legal notes
=================
| SPDX-FileCopyrightText: © 2022 ekvip automation GmbH <info@ekvip.de>
| SPDX-License-Identifier: Apache-2.0
| For details check: Apache-2.0_

.. _Apache-2.0: https://www.apache.org/licenses/LICENSE-2.0

.. </legal notes>



*)

METHOD orMaskIsEqualTo
VAR_INPUT
	(* current value to check *)
	currentValue	:__XWORD;
	(* 2nd operand for bitwise operation *)
	mask			:__XWORD;
	(* expected result after masking *)
	expectedValue	:__XWORD;
	(* message if the assertion is false *)
	message			:AssertMessage;
END_VAR
END_METHOD

(*

## Short summary
This assertion method checks if the result current value bitwise ``OR`` mask 
is not equal to the unexpected value

.. <legal notes>

legal notes
=================
| SPDX-FileCopyrightText: © 2022 ekvip automation GmbH <info@ekvip.de>
| SPDX-License-Identifier: Apache-2.0
| For details check: Apache-2.0_

.. _Apache-2.0: https://www.apache.org/licenses/LICENSE-2.0

.. </legal notes>



*)

METHOD orMaskIsNotEqualTo
VAR_INPUT
	(* current value to check *)
	currentValue	:__XWORD;
	(* 2nd operand for bitwise operation *)
	mask			:__XWORD;
	(* unexpected result after masking *)
	unexpectedValue	:__XWORD;
	(* message if the assertion is false *)
	message			:AssertMessage;
END_VAR
END_METHOD

(*

## Short summary
This assertion method checks if the current value is equal to the expected value

.. <legal notes>

legal notes
=================
| SPDX-FileCopyrightText: © 2022 ekvip automation GmbH <info@ekvip.de>
| SPDX-License-Identifier: Apache-2.0
| For details check: Apache-2.0_

.. _Apache-2.0: https://www.apache.org/licenses/LICENSE-2.0

.. </legal notes>



*)

METHOD valueIsEqualTo
VAR_INPUT
	(* current value to check *)
	currentValue	:__XWORD;
	(* expected value to compare *)
	expectedValue	:__XWORD;
	(* message if the assertion is false *)
	message			:AssertMessage;
END_VAR
END_METHOD

(*

## Short summary
This assertion method checks if the current value is greater than the less value

.. <legal notes>

legal notes
=================
| SPDX-FileCopyrightText: © 2022 ekvip automation GmbH <info@ekvip.de>
| SPDX-License-Identifier: Apache-2.0
| For details check: Apache-2.0_

.. _Apache-2.0: https://www.apache.org/licenses/LICENSE-2.0

.. </legal notes>



*)

METHOD valueIsGreaterThan
VAR_INPUT
	(* current value to check *)
	currentValue	:__XWORD;
	(* less than lower limit *)
	lessValue		:__XWORD;
	(* message if the assertion is false *)
	message			:AssertMessage;
END_VAR
END_METHOD

(*

## Short summary
This assertion method checks if the current value is inside a limit

**Attention:** 
	limits are included: ``valueIsInRangeOf(3, 3, 3)`` is a true assertion

.. <legal notes>

legal notes
=================
| SPDX-FileCopyrightText: © 2022 ekvip automation GmbH <info@ekvip.de>
| SPDX-License-Identifier: Apache-2.0
| For details check: Apache-2.0_

.. _Apache-2.0: https://www.apache.org/licenses/LICENSE-2.0

.. </legal notes>



*)

METHOD valueIsInRangeOf
VAR_INPUT
	(* lower limit for the current value *)
	lowerLimit		:__XWORD;
	(* current value to check *)
	currentValue	:__XWORD;
	(* upper limit for the current value *)
	upperLimit		:__XWORD;
	(* message if the assertion is false *)
	message			:AssertMessage;
END_VAR
END_METHOD

(*

## Short summary
This assertion method checks if the current value is less than the greater value

.. <legal notes>

legal notes
=================
| SPDX-FileCopyrightText: © 2022 ekvip automation GmbH <info@ekvip.de>
| SPDX-License-Identifier: Apache-2.0
| For details check: Apache-2.0_

.. _Apache-2.0: https://www.apache.org/licenses/LICENSE-2.0

.. </legal notes>



*)

METHOD valueIsLessThan
VAR_INPUT
	(* current value to check *)
	currentValue	:__XWORD;
	(* greater than upper limit *)
	greaterValue	:__XWORD;
	(* message if the assertion is false *)
	message			:AssertMessage;
END_VAR
END_METHOD

(*

## Short summary
This assertion method checks if the current value is less than or equal to the maximum value

.. <legal notes>

legal notes
=================
| SPDX-FileCopyrightText: © 2022 ekvip automation GmbH <info@ekvip.de>
| SPDX-License-Identifier: Apache-2.0
| For details check: Apache-2.0_

.. _Apache-2.0: https://www.apache.org/licenses/LICENSE-2.0

.. </legal notes>



*)

METHOD valueIsMax
VAR_INPUT
	(* current value to check *)
	currentValue	:__XWORD;
	(* upper limit for the current value *)
	maximumValue	:__XWORD;
	(* message if the assertion is false *)
	message			:AssertMessage;
END_VAR
END_METHOD

(*

## Short summary
This assertion method checks if the current value is greater than or equal to the minimum value

.. <legal notes>

legal notes
=================
| SPDX-FileCopyrightText: © 2022 ekvip automation GmbH <info@ekvip.de>
| SPDX-License-Identifier: Apache-2.0
| For details check: Apache-2.0_

.. _Apache-2.0: https://www.apache.org/licenses/LICENSE-2.0

.. </legal notes>



*)

METHOD valueIsMin
VAR_INPUT
	(* current value to check *)
	currentValue	:__XWORD;
	(* lower limit for the current value *)
	minimumValue	:__XWORD;
	(* message if the assertion is false *)
	message			:AssertMessage;
END_VAR
END_METHOD

(*

## Short summary
This assertion method checks if the current value is not equal to the unexpected value

.. <legal notes>

legal notes
=================
| SPDX-FileCopyrightText: © 2022 ekvip automation GmbH <info@ekvip.de>
| SPDX-License-Identifier: Apache-2.0
| For details check: Apache-2.0_

.. _Apache-2.0: https://www.apache.org/licenses/LICENSE-2.0

.. </legal notes>



*)

METHOD valueIsNotEqualTo
VAR_INPUT
	(* current value to check *)
	currentValue	:__XWORD;
	(* unexpected value to compare *)
	unexpectedValue	:__XWORD;
	(* message if the assertion is false *)
	message			:AssertMessage;
END_VAR
END_METHOD

(*

## Short summary
This assertion method checks if the result current value bitwise ``XOR`` mask is equal to the expected value

.. <legal notes>

legal notes
=================
| SPDX-FileCopyrightText: © 2022 ekvip automation GmbH <info@ekvip.de>
| SPDX-License-Identifier: Apache-2.0
| For details check: Apache-2.0_

.. _Apache-2.0: https://www.apache.org/licenses/LICENSE-2.0

.. </legal notes>



*)

METHOD xorMaskIsEqualTo
VAR_INPUT
	(* current value to check *)
	currentValue	:__XWORD;
	(* 2nd operand for bitwise operation *)
	mask			:__XWORD;
	(* expected result after masking *)
	expectedValue	:__XWORD;
	(* message if the assertion is false *)
	message			:AssertMessage;
END_VAR
END_METHOD

(*

## Short summary
This assertion method checks if the result current value bitwise ``XOR`` mask 
is not equal to the unexpected value

.. <legal notes>

legal notes
=================
| SPDX-FileCopyrightText: © 2022 ekvip automation GmbH <info@ekvip.de>
| SPDX-License-Identifier: Apache-2.0
| For details check: Apache-2.0_

.. _Apache-2.0: https://www.apache.org/licenses/LICENSE-2.0

.. </legal notes>



*)

METHOD xorMaskIsNotEqualTo
VAR_INPUT
	(* current value to check *)
	currentValue	:__XWORD;
	(* 2nd operand for bitwise operation *)
	mask			:__XWORD;
	(* unexpected result after masking *)
	unexpectedValue	:__XWORD;
	(* message if the assertion is false *)
	message			:AssertMessage;
END_VAR
END_METHOD

END_INTERFACE

// ---- Assertor/Assertions/BooleanAssertion/interfaces/IBooleanAssertion.TcIO
(*

## Short summary
This interface provides assert statements for booleans 

.. <legal notes>

legal notes
=================
| SPDX-FileCopyrightText: © 2022 ekvip automation GmbH <info@ekvip.de>
| SPDX-License-Identifier: Apache-2.0
| For details check: Apache-2.0_

.. _Apache-2.0: https://www.apache.org/licenses/LICENSE-2.0

.. </legal notes>



*)

INTERFACE IBooleanAssertion EXTENDS __SYSTEM.IQueryInterface

(*

## Short summary
This assertion method checks if the current value is equal to the expected value

.. <legal notes>

legal notes
=================
| SPDX-FileCopyrightText: © 2022 ekvip automation GmbH <info@ekvip.de>
| SPDX-License-Identifier: Apache-2.0
| For details check: Apache-2.0_

.. _Apache-2.0: https://www.apache.org/licenses/LICENSE-2.0

.. </legal notes>



*)

METHOD valueIsEqualTo
VAR_INPUT
	(* current value to check *)
	currentValue	:BOOL;
	(* expected value to compare *)
	expectedValue	:BOOL;
	(* message if the assertion is false *)
	message			:AssertMessage;
END_VAR
END_METHOD

(*

## Short summary
This assertion method checks if the current value is ``FALSE``

.. <legal notes>

legal notes
=================
| SPDX-FileCopyrightText: © 2022 ekvip automation GmbH <info@ekvip.de>
| SPDX-License-Identifier: Apache-2.0
| For details check: Apache-2.0_

.. _Apache-2.0: https://www.apache.org/licenses/LICENSE-2.0

.. </legal notes>



*)

METHOD valueIsFalse
VAR_INPUT
	(* current value to check *)
	currentValue	:BOOL;
	(* message if the assertion is false *)
	message			:AssertMessage;
END_VAR
END_METHOD

(*

## Short summary
This assertion method checks if the current value is not equal to the unexpected value

.. <legal notes>

legal notes
=================
| SPDX-FileCopyrightText: © 2022 ekvip automation GmbH <info@ekvip.de>
| SPDX-License-Identifier: Apache-2.0
| For details check: Apache-2.0_

.. _Apache-2.0: https://www.apache.org/licenses/LICENSE-2.0

.. </legal notes>



*)

METHOD valueIsNotEqualTo
VAR_INPUT
	(* current value to check *)
	currentValue	:BOOL;
	(* unexpected value to compare *)
	unexpectedValue	:BOOL;
	(* message if the assertion is false *)
	message			:AssertMessage;
END_VAR
END_METHOD

(*

## Short summary
This assertion method checks if the current value is ``TRUE``

.. <legal notes>

legal notes
=================
| SPDX-FileCopyrightText: © 2022 ekvip automation GmbH <info@ekvip.de>
| SPDX-License-Identifier: Apache-2.0
| For details check: Apache-2.0_

.. _Apache-2.0: https://www.apache.org/licenses/LICENSE-2.0

.. </legal notes>



*)

METHOD valueIsTrue
VAR_INPUT
	(* current value to check *)
	currentValue	:BOOL;
	(* message if the assertion is false *)
	message			:AssertMessage;
END_VAR
END_METHOD

END_INTERFACE

// ---- Assertor/Assertions/DateAndTimeAssertions/32Bit/Date/interfaces/I32BitDateAssertions.TcIO
(*

## Short summary
This interface provides assert statements for 32 bit ``DATE``  

.. <legal notes>

legal notes
=================
| SPDX-FileCopyrightText: © 2022 ekvip automation GmbH <info@ekvip.de>
| SPDX-License-Identifier: Apache-2.0
| For details check: Apache-2.0_

.. _Apache-2.0: https://www.apache.org/licenses/LICENSE-2.0

.. </legal notes>



*)

INTERFACE I32BitDateAssertions EXTENDS __SYSTEM.IQueryInterface

(*

## Short summary
This assertion method checks if the current value is equal to the expected value

.. <legal notes>

legal notes
=================
| SPDX-FileCopyrightText: © 2022 ekvip automation GmbH <info@ekvip.de>
| SPDX-License-Identifier: Apache-2.0
| For details check: Apache-2.0_

.. _Apache-2.0: https://www.apache.org/licenses/LICENSE-2.0

.. </legal notes>



*)

METHOD valueIsEqualTo
VAR_INPUT
	(* current value to check *)
	currentValue	:DATE;
	(* expected value to compare *)
	expectedValue	:DATE;
	(* message if the assertion is false *)
	message			:AssertMessage;
END_VAR
END_METHOD

(*

## Short summary
This assertion method checks if the current value is greater than the less value

.. <legal notes>

legal notes
=================
| SPDX-FileCopyrightText: © 2022 ekvip automation GmbH <info@ekvip.de>
| SPDX-License-Identifier: Apache-2.0
| For details check: Apache-2.0_

.. _Apache-2.0: https://www.apache.org/licenses/LICENSE-2.0

.. </legal notes>



*)

METHOD valueIsGreaterThan
VAR_INPUT
	(* current value to check *)
	currentValue	:DATE;
	(* less than lower limit *)
	lessValue		:DATE;
	(* message if the assertion is false *)
	message			:AssertMessage;
END_VAR
END_METHOD

(*

## Short summary
This assertion method checks if the current value is inside a limit

**Attention:** 
	limits are included: ``valueIsInRangeOf(date#1970-01-01, date#1970-01-01, date#1970-01-01)``
	is a true assertion

.. <legal notes>

legal notes
=================
| SPDX-FileCopyrightText: © 2022 ekvip automation GmbH <info@ekvip.de>
| SPDX-License-Identifier: Apache-2.0
| For details check: Apache-2.0_

.. _Apache-2.0: https://www.apache.org/licenses/LICENSE-2.0

.. </legal notes>



*)

METHOD valueIsInRangeOf
VAR_INPUT
	(* lower limit for the current value *)
	lowerLimit		:DATE;
	(* current value to check *)
	currentValue	:DATE;
	(* upper limit for the current value *)
	upperLimit		:DATE;
	(* message if the assertion is false *)
	message			:AssertMessage;
END_VAR
END_METHOD

(*

## Short summary
This assertion method checks if the current value is less than the greater value

.. <legal notes>

legal notes
=================
| SPDX-FileCopyrightText: © 2022 ekvip automation GmbH <info@ekvip.de>
| SPDX-License-Identifier: Apache-2.0
| For details check: Apache-2.0_

.. _Apache-2.0: https://www.apache.org/licenses/LICENSE-2.0

.. </legal notes>



*)

METHOD valueIsLessThan
VAR_INPUT
	(* current value to check *)
	currentValue	:DATE;
	(* greater than upper limit *)
	greaterValue	:DATE;
	(* message if the assertion is false *)
	message			:AssertMessage;
END_VAR
END_METHOD

(*

## Short summary
This assertion method checks if the current value is less than or equal to the maximum value

.. <legal notes>

legal notes
=================
| SPDX-FileCopyrightText: © 2022 ekvip automation GmbH <info@ekvip.de>
| SPDX-License-Identifier: Apache-2.0
| For details check: Apache-2.0_

.. _Apache-2.0: https://www.apache.org/licenses/LICENSE-2.0

.. </legal notes>



*)

METHOD valueIsMax
VAR_INPUT
	(* current value to check *)
	currentValue	:DATE;
	(* upper limit for the current value *)
	maximumValue	:DATE;
	(* message if the assertion is false *)
	message			:AssertMessage;
END_VAR
END_METHOD

(*

## Short summary
This assertion method checks if the current value is greater than or equal to the minimum value

.. <legal notes>

legal notes
=================
| SPDX-FileCopyrightText: © 2022 ekvip automation GmbH <info@ekvip.de>
| SPDX-License-Identifier: Apache-2.0
| For details check: Apache-2.0_

.. _Apache-2.0: https://www.apache.org/licenses/LICENSE-2.0

.. </legal notes>



*)

METHOD valueIsMin
VAR_INPUT
	(* current value to check *)
	currentValue	:DATE;
	(* lower limit for the current value *)
	minimumValue	:DATE;
	(* message if the assertion is false *)
	message			:AssertMessage;
END_VAR
END_METHOD

(*

## Short summary
This assertion method checks if the current value is not equal to the unexpected value

.. <legal notes>

legal notes
=================
| SPDX-FileCopyrightText: © 2022 ekvip automation GmbH <info@ekvip.de>
| SPDX-License-Identifier: Apache-2.0
| For details check: Apache-2.0_

.. _Apache-2.0: https://www.apache.org/licenses/LICENSE-2.0

.. </legal notes>



*)

METHOD valueIsNotEqualTo
VAR_INPUT
	(* current value to check *)
	currentValue	:DATE;
	(* unexpected value to compare *)
	unexpectedValue	:DATE;
	(* message if the assertion is false *)
	message			:AssertMessage;
END_VAR
END_METHOD

END_INTERFACE

// ---- Assertor/Assertions/DateAndTimeAssertions/32Bit/DT/interfaces/I32BitDtAssertions.TcIO
(*

## Short summary
This interface provides assert statements for 32 bit date and time ``DT``  

.. <legal notes>

legal notes
=================
| SPDX-FileCopyrightText: © 2022 ekvip automation GmbH <info@ekvip.de>
| SPDX-License-Identifier: Apache-2.0
| For details check: Apache-2.0_

.. _Apache-2.0: https://www.apache.org/licenses/LICENSE-2.0

.. </legal notes>



*)

INTERFACE I32BitDtAssertions EXTENDS __SYSTEM.IQueryInterface

(*

## Short summary
This assertion method checks if the current value is equal to the expected value

.. <legal notes>

legal notes
=================
| SPDX-FileCopyrightText: © 2022 ekvip automation GmbH <info@ekvip.de>
| SPDX-License-Identifier: Apache-2.0
| For details check: Apache-2.0_

.. _Apache-2.0: https://www.apache.org/licenses/LICENSE-2.0

.. </legal notes>



*)

METHOD valueIsEqualTo
VAR_INPUT
	(* current value to check *)
	currentValue	:DT;
	(* expected value to compare *)
	expectedValue	:DT;
	(* message if the assertion is false *)
	message			:AssertMessage;
END_VAR
END_METHOD

(*

## Short summary
This assertion method checks if the current value is greater than the less value

.. <legal notes>

legal notes
=================
| SPDX-FileCopyrightText: © 2022 ekvip automation GmbH <info@ekvip.de>
| SPDX-License-Identifier: Apache-2.0
| For details check: Apache-2.0_

.. _Apache-2.0: https://www.apache.org/licenses/LICENSE-2.0

.. </legal notes>



*)

METHOD valueIsGreaterThan
VAR_INPUT
	(* current value to check *)
	currentValue	:DT;
	(* less than lower limit *)
	lessValue		:DT;
	(* message if the assertion is false *)
	message			:AssertMessage;
END_VAR
END_METHOD

(*

## Short summary
This assertion method checks if the current value is inside a limit

**Attention:** 
	limits are included: ``valueIsInRangeOf(dt#1970-01-01-0:0:0, dt#1970-01-01-0:0:0, dt#1970-01-01-0:0:0)``
	is a true assertion

.. <legal notes>

legal notes
=================
| SPDX-FileCopyrightText: © 2022 ekvip automation GmbH <info@ekvip.de>
| SPDX-License-Identifier: Apache-2.0
| For details check: Apache-2.0_

.. _Apache-2.0: https://www.apache.org/licenses/LICENSE-2.0

.. </legal notes>



*)

METHOD valueIsInRangeOf
VAR_INPUT
	(* lower limit for the current value *)
	lowerLimit		:DT;
	(* current value to check *)
	currentValue	:DT;
	(* upper limit for the current value *)
	upperLimit		:DT;
	(* message if the assertion is false *)
	message			:AssertMessage;
END_VAR
END_METHOD

(*

## Short summary
This assertion method checks if the current value is less than the greater value

.. <legal notes>

legal notes
=================
| SPDX-FileCopyrightText: © 2022 ekvip automation GmbH <info@ekvip.de>
| SPDX-License-Identifier: Apache-2.0
| For details check: Apache-2.0_

.. _Apache-2.0: https://www.apache.org/licenses/LICENSE-2.0

.. </legal notes>



*)

METHOD valueIsLessThan
VAR_INPUT
	(* current value to check *)
	currentValue	:DT;
	(* greater than upper limit *)
	greaterValue	:DT;
	(* message if the assertion is false *)
	message			:AssertMessage;
END_VAR
END_METHOD

(*

## Short summary
This assertion method checks if the current value is less than or equal to the maximum value

.. <legal notes>

legal notes
=================
| SPDX-FileCopyrightText: © 2022 ekvip automation GmbH <info@ekvip.de>
| SPDX-License-Identifier: Apache-2.0
| For details check: Apache-2.0_

.. _Apache-2.0: https://www.apache.org/licenses/LICENSE-2.0

.. </legal notes>



*)

METHOD valueIsMax
VAR_INPUT
	(* current value to check *)
	currentValue	:DT;
	(* upper limit for the current value *)
	maximumValue	:DT;
	(* message if the assertion is false *)
	message			:AssertMessage;
END_VAR
END_METHOD

(*

## Short summary
This assertion method checks if the current value is greater than or equal to the minimum value

.. <legal notes>

legal notes
=================
| SPDX-FileCopyrightText: © 2022 ekvip automation GmbH <info@ekvip.de>
| SPDX-License-Identifier: Apache-2.0
| For details check: Apache-2.0_

.. _Apache-2.0: https://www.apache.org/licenses/LICENSE-2.0

.. </legal notes>



*)

METHOD valueIsMin
VAR_INPUT
	(* current value to check *)
	currentValue	:DT;
	(* lower limit for the current value *)
	minimumValue	:DT;
	(* message if the assertion is false *)
	message			:AssertMessage;
END_VAR
END_METHOD

(*

## Short summary
This assertion method checks if the current value is not equal to the unexpected value

.. <legal notes>

legal notes
=================
| SPDX-FileCopyrightText: © 2022 ekvip automation GmbH <info@ekvip.de>
| SPDX-License-Identifier: Apache-2.0
| For details check: Apache-2.0_

.. _Apache-2.0: https://www.apache.org/licenses/LICENSE-2.0

.. </legal notes>



*)

METHOD valueIsNotEqualTo
VAR_INPUT
	(* current value to check *)
	currentValue	:DT;
	(* unexpected value to compare *)
	unexpectedValue	:DT;
	(* message if the assertion is false *)
	message			:AssertMessage;
END_VAR
END_METHOD

END_INTERFACE

// ---- Assertor/Assertions/DateAndTimeAssertions/32Bit/interfaces/ISimpleDateAndTimeAssertions.TcIO
(*

## Short summary

This interface provides assert statements for date and time types with 32 bit length
For date and time (``DT``) use `ISimpleDateAndTimeAssertions.dateAndTime`
For date (``DATE``) use  `ISimpleDateAndTimeAssertions.dateOnly`
For time of day (``TOD``) use  `ISimpleDateAndTimeAssertions.timeOfDay`

.. <legal notes>

legal notes
=================
| SPDX-FileCopyrightText: © 2022 ekvip automation GmbH <info@ekvip.de>
| SPDX-License-Identifier: Apache-2.0
| For details check: Apache-2.0_

.. _Apache-2.0: https://www.apache.org/licenses/LICENSE-2.0

.. </legal notes>



*)

INTERFACE ISimpleDateAndTimeAssertions EXTENDS __SYSTEM.IQueryInterface

(*

## Short summary
Returns the interface `I32BitDtAssertions` with assert statements for 32 bit date and time ``DT``

.. <legal notes>

legal notes
=================
| SPDX-FileCopyrightText: © 2022 ekvip automation GmbH <info@ekvip.de>
| SPDX-License-Identifier: Apache-2.0
| For details check: Apache-2.0_

.. _Apache-2.0: https://www.apache.org/licenses/LICENSE-2.0

.. </legal notes>

*)

PROPERTY dateAndTime :I32BitDtAssertions
GET
END_GET
END_PROPERTY

(*

## Short summary
Returns the interface `I32BitDateAssertions` with assert statements for 32 bit date ``DATE``

.. <legal notes>

legal notes
=================
| SPDX-FileCopyrightText: © 2022 ekvip automation GmbH <info@ekvip.de>
| SPDX-License-Identifier: Apache-2.0
| For details check: Apache-2.0_

.. _Apache-2.0: https://www.apache.org/licenses/LICENSE-2.0

.. </legal notes>

*)

PROPERTY dateOnly :I32BitDateAssertions
GET
END_GET
END_PROPERTY

(*

## Short summary
Returns the interface `I32BitTodAssertions` with assert statements for 32 bit time of day ``TOD``

.. <legal notes>

legal notes
=================
| SPDX-FileCopyrightText: © 2022 ekvip automation GmbH <info@ekvip.de>
| SPDX-License-Identifier: Apache-2.0
| For details check: Apache-2.0_

.. _Apache-2.0: https://www.apache.org/licenses/LICENSE-2.0

.. </legal notes>

*)

PROPERTY timeOfDay :I32BitTodAssertions
GET
END_GET
END_PROPERTY

END_INTERFACE

// ---- Assertor/Assertions/DateAndTimeAssertions/32Bit/TOD/interfaces/I32BitTodAssertions.TcIO
(*

## Short summary
This interface provides assert statements for 32 bit time of day ``TOD``  

.. <legal notes>

legal notes
=================
| SPDX-FileCopyrightText: © 2022 ekvip automation GmbH <info@ekvip.de>
| SPDX-License-Identifier: Apache-2.0
| For details check: Apache-2.0_

.. _Apache-2.0: https://www.apache.org/licenses/LICENSE-2.0

.. </legal notes>



*)

INTERFACE I32BitTodAssertions EXTENDS __SYSTEM.IQueryInterface

(*

## Short summary
This assertion method checks if the current value is equal to the expected value

.. <legal notes>

legal notes
=================
| SPDX-FileCopyrightText: © 2022 ekvip automation GmbH <info@ekvip.de>
| SPDX-License-Identifier: Apache-2.0
| For details check: Apache-2.0_

.. _Apache-2.0: https://www.apache.org/licenses/LICENSE-2.0

.. </legal notes>



*)

METHOD valueIsEqualTo
VAR_INPUT
	(* current value to check *)
	currentValue	:TOD;
	(* expected value to compare *)
	expectedValue	:TOD;
	(* message if the assertion is false *)
	message			:AssertMessage;
END_VAR
END_METHOD

(*

## Short summary
This assertion method checks if the current value is greater than the less value

.. <legal notes>

legal notes
=================
| SPDX-FileCopyrightText: © 2022 ekvip automation GmbH <info@ekvip.de>
| SPDX-License-Identifier: Apache-2.0
| For details check: Apache-2.0_

.. _Apache-2.0: https://www.apache.org/licenses/LICENSE-2.0

.. </legal notes>



*)

METHOD valueIsGreaterThan
VAR_INPUT
	(* current value to check *)
	currentValue	:TOD;
	(* less than lower limit *)
	lessValue		:TOD;
	(* message if the assertion is false *)
	message			:AssertMessage;
END_VAR
END_METHOD

(*

## Short summary
This assertion method checks if the current value is inside a limit

**Attention:** 
	limits are included: ``valueIsInRangeOf(tod#3:0:0, tod#3:0:0, tod#3:0:0)`` is a true assertion

.. <legal notes>

legal notes
=================
| SPDX-FileCopyrightText: © 2022 ekvip automation GmbH <info@ekvip.de>
| SPDX-License-Identifier: Apache-2.0
| For details check: Apache-2.0_

.. _Apache-2.0: https://www.apache.org/licenses/LICENSE-2.0

.. </legal notes>



*)

METHOD valueIsInRangeOf
VAR_INPUT
	(* lower limit for the current value *)
	lowerLimit		:TOD;
	(* current value to check *)
	currentValue	:TOD;
	(* upper limit for the current value *)
	upperLimit		:TOD;
	(* message if the assertion is false *)
	message			:AssertMessage;
END_VAR
END_METHOD

(*

## Short summary
This assertion method checks if the current value is less than the greater value

.. <legal notes>

legal notes
=================
| SPDX-FileCopyrightText: © 2022 ekvip automation GmbH <info@ekvip.de>
| SPDX-License-Identifier: Apache-2.0
| For details check: Apache-2.0_

.. _Apache-2.0: https://www.apache.org/licenses/LICENSE-2.0

.. </legal notes>



*)

METHOD valueIsLessThan
VAR_INPUT
	(* current value to check *)
	currentValue	:TOD;
	(* greater than upper limit *)
	greaterValue	:TOD;
	(* message if the assertion is false *)
	message			:AssertMessage;
END_VAR
END_METHOD

(*

## Short summary
This assertion method checks if the current value is less than or equal to the maximum value

.. <legal notes>

legal notes
=================
| SPDX-FileCopyrightText: © 2022 ekvip automation GmbH <info@ekvip.de>
| SPDX-License-Identifier: Apache-2.0
| For details check: Apache-2.0_

.. _Apache-2.0: https://www.apache.org/licenses/LICENSE-2.0

.. </legal notes>



*)

METHOD valueIsMax
VAR_INPUT
	(* current value to check *)
	currentValue	:TOD;
	(* upper limit for the current value *)
	maximumValue	:TOD;
	(* message if the assertion is false *)
	message			:AssertMessage;
END_VAR
END_METHOD

(*

## Short summary
This assertion method checks if the current value is greater than or equal to the minimum value

.. <legal notes>

legal notes
=================
| SPDX-FileCopyrightText: © 2022 ekvip automation GmbH <info@ekvip.de>
| SPDX-License-Identifier: Apache-2.0
| For details check: Apache-2.0_

.. _Apache-2.0: https://www.apache.org/licenses/LICENSE-2.0

.. </legal notes>



*)

METHOD valueIsMin
VAR_INPUT
	(* current value to check *)
	currentValue	:TOD;
	(* lower limit for the current value *)
	minimumValue	:TOD;
	(* message if the assertion is false *)
	message			:AssertMessage;
END_VAR
END_METHOD

(*

## Short summary
This assertion method checks if the current value is not equal to the unexpected value

.. <legal notes>

legal notes
=================
| SPDX-FileCopyrightText: © 2022 ekvip automation GmbH <info@ekvip.de>
| SPDX-License-Identifier: Apache-2.0
| For details check: Apache-2.0_

.. _Apache-2.0: https://www.apache.org/licenses/LICENSE-2.0

.. </legal notes>



*)

METHOD valueIsNotEqualTo
VAR_INPUT
	(* current value to check *)
	currentValue	:TOD;
	(* unexpected value to compare *)
	unexpectedValue	:TOD;
	(* message if the assertion is false *)
	message			:AssertMessage;
END_VAR
END_METHOD

END_INTERFACE

// ---- Assertor/Assertions/DateAndTimeAssertions/64Bit/LDate/interfaces/I64BitDateAssertions.TcIO
(*

## Short summary
This interface provides assert statements for 32 bit ``DATE``  

.. <legal notes>

legal notes
=================
| SPDX-FileCopyrightText: © 2022 ekvip automation GmbH <info@ekvip.de>
| SPDX-License-Identifier: Apache-2.0
| For details check: Apache-2.0_

.. _Apache-2.0: https://www.apache.org/licenses/LICENSE-2.0

.. </legal notes>



*)

INTERFACE I64BitDateAssertions EXTENDS __SYSTEM.IQueryInterface

(*

## Short summary
This assertion method checks if the current value is equal to the expected value

.. <legal notes>

legal notes
=================
| SPDX-FileCopyrightText: © 2022 ekvip automation GmbH <info@ekvip.de>
| SPDX-License-Identifier: Apache-2.0
| For details check: Apache-2.0_

.. _Apache-2.0: https://www.apache.org/licenses/LICENSE-2.0

.. </legal notes>



*)

METHOD valueIsEqualTo
VAR_INPUT
	(* current value to check *)
	currentValue	:LDATE;
	(* expected value to compare *)
	expectedValue	:LDATE;
	(* message if the assertion is false *)
	message			:AssertMessage;
END_VAR
END_METHOD

(*

## Short summary
This assertion method checks if the current value is greater than the less value

.. <legal notes>

legal notes
=================
| SPDX-FileCopyrightText: © 2022 ekvip automation GmbH <info@ekvip.de>
| SPDX-License-Identifier: Apache-2.0
| For details check: Apache-2.0_

.. _Apache-2.0: https://www.apache.org/licenses/LICENSE-2.0

.. </legal notes>



*)

METHOD valueIsGreaterThan
VAR_INPUT
	(* current value to check *)
	currentValue	:LDATE;
	(* less than lower limit *)
	lessValue		:LDATE;
	(* message if the assertion is false *)
	message			:AssertMessage;
END_VAR
END_METHOD

(*

## Short summary
This assertion method checks if the current value is inside a limit

**Attention:** 
	limits are included: ``valueIsInRangeOf(ldate#1970-01-01, ldate#1970-01-01, ldate#1970-01-01)``
	is a true assertion

.. <legal notes>

legal notes
=================
| SPDX-FileCopyrightText: © 2022 ekvip automation GmbH <info@ekvip.de>
| SPDX-License-Identifier: Apache-2.0
| For details check: Apache-2.0_

.. _Apache-2.0: https://www.apache.org/licenses/LICENSE-2.0

.. </legal notes>



*)

METHOD valueIsInRangeOf
VAR_INPUT
	(* lower limit for the current value *)
	lowerLimit		:LDATE;
	(* current value to check *)
	currentValue	:LDATE;
	(* upper limit for the current value *)
	upperLimit		:LDATE;
	(* message if the assertion is false *)
	message			:AssertMessage;
END_VAR
END_METHOD

(*

## Short summary
This assertion method checks if the current value is less than the greater value

.. <legal notes>

legal notes
=================
| SPDX-FileCopyrightText: © 2022 ekvip automation GmbH <info@ekvip.de>
| SPDX-License-Identifier: Apache-2.0
| For details check: Apache-2.0_

.. _Apache-2.0: https://www.apache.org/licenses/LICENSE-2.0

.. </legal notes>



*)

METHOD valueIsLessThan
VAR_INPUT
	(* current value to check *)
	currentValue	:LDATE;
	(* greater than upper limit *)
	greaterValue	:LDATE;
	(* message if the assertion is false *)
	message			:AssertMessage;
END_VAR
END_METHOD

(*

## Short summary
This assertion method checks if the current value is less than or equal to the maximum value

.. <legal notes>

legal notes
=================
| SPDX-FileCopyrightText: © 2022 ekvip automation GmbH <info@ekvip.de>
| SPDX-License-Identifier: Apache-2.0
| For details check: Apache-2.0_

.. _Apache-2.0: https://www.apache.org/licenses/LICENSE-2.0

.. </legal notes>



*)

METHOD valueIsMax
VAR_INPUT
	(* current value to check *)
	currentValue	:LDATE;
	(* upper limit for the current value *)
	maximumValue	:LDATE;
	(* message if the assertion is false *)
	message			:AssertMessage;
END_VAR
END_METHOD

(*

## Short summary
This assertion method checks if the current value is greater than or equal to the minimum value

.. <legal notes>

legal notes
=================
| SPDX-FileCopyrightText: © 2022 ekvip automation GmbH <info@ekvip.de>
| SPDX-License-Identifier: Apache-2.0
| For details check: Apache-2.0_

.. _Apache-2.0: https://www.apache.org/licenses/LICENSE-2.0

.. </legal notes>



*)

METHOD valueIsMin
VAR_INPUT
	(* current value to check *)
	currentValue	:LDATE;
	(* lower limit for the current value *)
	minimumValue	:LDATE;
	(* message if the assertion is false *)
	message			:AssertMessage;
END_VAR
END_METHOD

(*

## Short summary
This assertion method checks if the current value is not equal to the unexpected value

.. <legal notes>

legal notes
=================
| SPDX-FileCopyrightText: © 2022 ekvip automation GmbH <info@ekvip.de>
| SPDX-License-Identifier: Apache-2.0
| For details check: Apache-2.0_

.. _Apache-2.0: https://www.apache.org/licenses/LICENSE-2.0

.. </legal notes>



*)

METHOD valueIsNotEqualTo
VAR_INPUT
	(* current value to check *)
	currentValue	:LDATE;
	(* unexpected value to compare *)
	unexpectedValue	:LDATE;
	(* message if the assertion is false *)
	message			:AssertMessage;
END_VAR
END_METHOD

END_INTERFACE

// ---- Assertor/Assertions/DateAndTimeAssertions/64Bit/LDT/interfaces/I64BitDtAssertions.TcIO
(*

## Short summary
This interface provides assert statements for 64 bit date and time ``LDT``  

.. <legal notes>

legal notes
=================
| SPDX-FileCopyrightText: © 2022 ekvip automation GmbH <info@ekvip.de>
| SPDX-License-Identifier: Apache-2.0
| For details check: Apache-2.0_

.. _Apache-2.0: https://www.apache.org/licenses/LICENSE-2.0

.. </legal notes>



*)

INTERFACE I64BitDtAssertions EXTENDS __SYSTEM.IQueryInterface

(*

## Short summary
This assertion method checks if the current value is equal to the expected value

.. <legal notes>

legal notes
=================
| SPDX-FileCopyrightText: © 2022 ekvip automation GmbH <info@ekvip.de>
| SPDX-License-Identifier: Apache-2.0
| For details check: Apache-2.0_

.. _Apache-2.0: https://www.apache.org/licenses/LICENSE-2.0

.. </legal notes>



*)

METHOD valueIsEqualTo
VAR_INPUT
	(* current value to check *)
	currentValue	:LDT;
	(* expected value to compare *)
	expectedValue	:LDT;
	(* message if the assertion is false *)
	message			:AssertMessage;
END_VAR
END_METHOD

(*

## Short summary
This assertion method checks if the current value is greater than the less value

.. <legal notes>

legal notes
=================
| SPDX-FileCopyrightText: © 2022 ekvip automation GmbH <info@ekvip.de>
| SPDX-License-Identifier: Apache-2.0
| For details check: Apache-2.0_

.. _Apache-2.0: https://www.apache.org/licenses/LICENSE-2.0

.. </legal notes>



*)

METHOD valueIsGreaterThan
VAR_INPUT
	(* current value to check *)
	currentValue	:LDT;
	(* less than lower limit *)
	lessValue		:LDT;
	(* message if the assertion is false *)
	message			:AssertMessage;
END_VAR
END_METHOD

(*

## Short summary
This assertion method checks if the current value is inside a limit

**Attention:** 
	limits are included: ``valueIsInRangeOf(ldt#1970-01-01-0:0:0, ldt#1970-01-01-0:0:0, ldt#1970-01-01-0:0:0)``
	is a true assertion

.. <legal notes>

legal notes
=================
| SPDX-FileCopyrightText: © 2022 ekvip automation GmbH <info@ekvip.de>
| SPDX-License-Identifier: Apache-2.0
| For details check: Apache-2.0_

.. _Apache-2.0: https://www.apache.org/licenses/LICENSE-2.0

.. </legal notes>



*)

METHOD valueIsInRangeOf
VAR_INPUT
	(* lower limit for the current value *)
	lowerLimit		:LDT;
	(* current value to check *)
	currentValue	:LDT;
	(* upper limit for the current value *)
	upperLimit		:LDT;
	(* message if the assertion is false *)
	message			:AssertMessage;
END_VAR
END_METHOD

(*

## Short summary
This assertion method checks if the current value is less than the greater value

.. <legal notes>

legal notes
=================
| SPDX-FileCopyrightText: © 2022 ekvip automation GmbH <info@ekvip.de>
| SPDX-License-Identifier: Apache-2.0
| For details check: Apache-2.0_

.. _Apache-2.0: https://www.apache.org/licenses/LICENSE-2.0

.. </legal notes>



*)

METHOD valueIsLessThan
VAR_INPUT
	(* current value to check *)
	currentValue	:LDT;
	(* greater than upper limit *)
	greaterValue	:LDT;
	(* message if the assertion is false *)
	message			:AssertMessage;
END_VAR
END_METHOD

(*

## Short summary
This assertion method checks if the current value is less than or equal to the maximum value

.. <legal notes>

legal notes
=================
| SPDX-FileCopyrightText: © 2022 ekvip automation GmbH <info@ekvip.de>
| SPDX-License-Identifier: Apache-2.0
| For details check: Apache-2.0_

.. _Apache-2.0: https://www.apache.org/licenses/LICENSE-2.0

.. </legal notes>



*)

METHOD valueIsMax
VAR_INPUT
	(* current value to check *)
	currentValue	:LDT;
	(* upper limit for the current value *)
	maximumValue	:LDT;
	(* message if the assertion is false *)
	message			:AssertMessage;
END_VAR
END_METHOD

(*

## Short summary
This assertion method checks if the current value is greater than or equal to the minimum value

.. <legal notes>

legal notes
=================
| SPDX-FileCopyrightText: © 2022 ekvip automation GmbH <info@ekvip.de>
| SPDX-License-Identifier: Apache-2.0
| For details check: Apache-2.0_

.. _Apache-2.0: https://www.apache.org/licenses/LICENSE-2.0

.. </legal notes>



*)

METHOD valueIsMin
VAR_INPUT
	(* current value to check *)
	currentValue	:LDT;
	(* lower limit for the current value *)
	minimumValue	:LDT;
	(* message if the assertion is false *)
	message			:AssertMessage;
END_VAR
END_METHOD

(*

## Short summary
This assertion method checks if the current value is not equal to the unexpected value

.. <legal notes>

legal notes
=================
| SPDX-FileCopyrightText: © 2022 ekvip automation GmbH <info@ekvip.de>
| SPDX-License-Identifier: Apache-2.0
| For details check: Apache-2.0_

.. _Apache-2.0: https://www.apache.org/licenses/LICENSE-2.0

.. </legal notes>



*)

METHOD valueIsNotEqualTo
VAR_INPUT
	(* current value to check *)
	currentValue	:LDT;
	(* unexpected value to compare *)
	unexpectedValue	:LDT;
	(* message if the assertion is false *)
	message			:AssertMessage;
END_VAR
END_METHOD

END_INTERFACE

// ---- Assertor/Assertions/DateAndTimeAssertions/64Bit/interfaces/ILongDateAndTimeAssertions.TcIO
(*

## Short summary

This interface provides assert statements for date and time types with 64 bit length
For date and time (``LDT``) use `ISimpleDateAndTimeAssertions.dateAndTime`
For date (``LDATE``) use  `ISimpleDateAndTimeAssertions.dateOnly`
For time of day (``LTOD``) use  `ISimpleDateAndTimeAssertions.timeOfDay`

.. <legal notes>

legal notes
=================
| SPDX-FileCopyrightText: © 2022 ekvip automation GmbH <info@ekvip.de>
| SPDX-License-Identifier: Apache-2.0
| For details check: Apache-2.0_

.. _Apache-2.0: https://www.apache.org/licenses/LICENSE-2.0

.. </legal notes>



*)

INTERFACE ILongDateAndTimeAssertions EXTENDS __SYSTEM.IQueryInterface

(*

## Short summary
Returns the interface `I64BitDtAssertions` with assert statements for 64 bit date and time ``LDT``

.. <legal notes>

legal notes
=================
| SPDX-FileCopyrightText: © 2022 ekvip automation GmbH <info@ekvip.de>
| SPDX-License-Identifier: Apache-2.0
| For details check: Apache-2.0_

.. _Apache-2.0: https://www.apache.org/licenses/LICENSE-2.0

.. </legal notes>

*)

PROPERTY dateAndTime :I64BitDtAssertions
GET
END_GET
END_PROPERTY

(*

## Short summary
Returns the interface `I64BitDateAssertions` with assert statements for 64 bit date ``LDATE``

.. <legal notes>

legal notes
=================
| SPDX-FileCopyrightText: © 2022 ekvip automation GmbH <info@ekvip.de>
| SPDX-License-Identifier: Apache-2.0
| For details check: Apache-2.0_

.. _Apache-2.0: https://www.apache.org/licenses/LICENSE-2.0

.. </legal notes>

*)

PROPERTY dateOnly :I64BitDateAssertions
GET
END_GET
END_PROPERTY

(*

## Short summary
Returns the interface `I64BitTodAssertions` with assert statements for 32 bit time of day ``LTOD``

.. <legal notes>

legal notes
=================
| SPDX-FileCopyrightText: © 2022 ekvip automation GmbH <info@ekvip.de>
| SPDX-License-Identifier: Apache-2.0
| For details check: Apache-2.0_

.. _Apache-2.0: https://www.apache.org/licenses/LICENSE-2.0

.. </legal notes>

*)

PROPERTY timeOfDay :I64BitTodAssertions
GET
END_GET
END_PROPERTY

END_INTERFACE

// ---- Assertor/Assertions/DateAndTimeAssertions/64Bit/LTOD/interfaces/I64BitTodAssertions.TcIO
(*

## Short summary
This interface provides assert statements for 64 bit time of day ``LTOD``  

.. <legal notes>

legal notes
=================
| SPDX-FileCopyrightText: © 2022 ekvip automation GmbH <info@ekvip.de>
| SPDX-License-Identifier: Apache-2.0
| For details check: Apache-2.0_

.. _Apache-2.0: https://www.apache.org/licenses/LICENSE-2.0

.. </legal notes>



*)

INTERFACE I64BitTodAssertions EXTENDS __SYSTEM.IQueryInterface

(*

## Short summary
This assertion method checks if the current value is equal to the expected value

.. <legal notes>

legal notes
=================
| SPDX-FileCopyrightText: © 2022 ekvip automation GmbH <info@ekvip.de>
| SPDX-License-Identifier: Apache-2.0
| For details check: Apache-2.0_

.. _Apache-2.0: https://www.apache.org/licenses/LICENSE-2.0

.. </legal notes>



*)

METHOD valueIsEqualTo
VAR_INPUT
	(* current value to check *)
	currentValue	:LTOD;
	(* expected value to compare *)
	expectedValue	:LTOD;
	(* message if the assertion is false *)
	message			:AssertMessage;
END_VAR
END_METHOD

(*

## Short summary
This assertion method checks if the current value is greater than the less value

.. <legal notes>

legal notes
=================
| SPDX-FileCopyrightText: © 2022 ekvip automation GmbH <info@ekvip.de>
| SPDX-License-Identifier: Apache-2.0
| For details check: Apache-2.0_

.. _Apache-2.0: https://www.apache.org/licenses/LICENSE-2.0

.. </legal notes>



*)

METHOD valueIsGreaterThan
VAR_INPUT
	(* current value to check *)
	currentValue	:LTOD;
	(* less than lower limit *)
	lessValue		:LTOD;
	(* message if the assertion is false *)
	message			:AssertMessage;
END_VAR
END_METHOD

(*

## Short summary
This assertion method checks if the current value is inside a limit

**Attention:** 
	limits are included: ``valueIsInRangeOf(ltod#3:0:0, ltod#3:0:0, ltod#3:0:0)`` is a true assertion

.. <legal notes>

legal notes
=================
| SPDX-FileCopyrightText: © 2022 ekvip automation GmbH <info@ekvip.de>
| SPDX-License-Identifier: Apache-2.0
| For details check: Apache-2.0_

.. _Apache-2.0: https://www.apache.org/licenses/LICENSE-2.0

.. </legal notes>



*)

METHOD valueIsInRangeOf
VAR_INPUT
	(* lower limit for the current value *)
	lowerLimit		:LTOD;
	(* current value to check *)
	currentValue	:LTOD;
	(* upper limit for the current value *)
	upperLimit		:LTOD;
	(* message if the assertion is false *)
	message			:AssertMessage;
END_VAR
END_METHOD

(*

## Short summary
This assertion method checks if the current value is less than the greater value

.. <legal notes>

legal notes
=================
| SPDX-FileCopyrightText: © 2022 ekvip automation GmbH <info@ekvip.de>
| SPDX-License-Identifier: Apache-2.0
| For details check: Apache-2.0_

.. _Apache-2.0: https://www.apache.org/licenses/LICENSE-2.0

.. </legal notes>



*)

METHOD valueIsLessThan
VAR_INPUT
	(* current value to check *)
	currentValue	:LTOD;
	(* greater than upper limit *)
	greaterValue	:LTOD;
	(* message if the assertion is false *)
	message			:AssertMessage;
END_VAR
END_METHOD

(*

## Short summary
This assertion method checks if the current value is less than or equal to the maximum value

.. <legal notes>

legal notes
=================
| SPDX-FileCopyrightText: © 2022 ekvip automation GmbH <info@ekvip.de>
| SPDX-License-Identifier: Apache-2.0
| For details check: Apache-2.0_

.. _Apache-2.0: https://www.apache.org/licenses/LICENSE-2.0

.. </legal notes>



*)

METHOD valueIsMax
VAR_INPUT
	(* current value to check *)
	currentValue	:LTOD;
	(* upper limit for the current value *)
	maximumValue	:LTOD;
	(* message if the assertion is false *)
	message			:AssertMessage;
END_VAR
END_METHOD

(*

## Short summary
This assertion method checks if the current value is greater than or equal to the minimum value

.. <legal notes>

legal notes
=================
| SPDX-FileCopyrightText: © 2022 ekvip automation GmbH <info@ekvip.de>
| SPDX-License-Identifier: Apache-2.0
| For details check: Apache-2.0_

.. _Apache-2.0: https://www.apache.org/licenses/LICENSE-2.0

.. </legal notes>



*)

METHOD valueIsMin
VAR_INPUT
	(* current value to check *)
	currentValue	:LTOD;
	(* lower limit for the current value *)
	minimumValue	:LTOD;
	(* message if the assertion is false *)
	message			:AssertMessage;
END_VAR
END_METHOD

(*

## Short summary
This assertion method checks if the current value is not equal to the unexpected value

.. <legal notes>

legal notes
=================
| SPDX-FileCopyrightText: © 2022 ekvip automation GmbH <info@ekvip.de>
| SPDX-License-Identifier: Apache-2.0
| For details check: Apache-2.0_

.. _Apache-2.0: https://www.apache.org/licenses/LICENSE-2.0

.. </legal notes>



*)

METHOD valueIsNotEqualTo
VAR_INPUT
	(* current value to check *)
	currentValue	:LTOD;
	(* unexpected value to compare *)
	unexpectedValue	:LTOD;
	(* message if the assertion is false *)
	message			:AssertMessage;
END_VAR
END_METHOD

END_INTERFACE

// ---- Assertor/Assertions/DateAndTimeAssertions/interfaces/IDateAndTimeAssertions.TcIO
(*

## Short summary

This interface provides assert statements for date and time types
For 32 bit date and time types use `IDateAndTimeAssertions.simple`
For 64 bit date and time types use `IDateAndTimeAssertions.long`

.. <legal notes>

legal notes
=================
| SPDX-FileCopyrightText: © 2022 ekvip automation GmbH <info@ekvip.de>
| SPDX-License-Identifier: Apache-2.0
| For details check: Apache-2.0_

.. _Apache-2.0: https://www.apache.org/licenses/LICENSE-2.0

.. </legal notes>



*)

INTERFACE IDateAndTimeAssertions EXTENDS __SYSTEM.IQueryInterface

(*

## Short summary
Returns an interface with assert statements for 64 bit times 

.. <legal notes>

legal notes
=================
| SPDX-FileCopyrightText: © 2022 ekvip automation GmbH <info@ekvip.de>
| SPDX-License-Identifier: Apache-2.0
| For details check: Apache-2.0_

.. _Apache-2.0: https://www.apache.org/licenses/LICENSE-2.0

.. </legal notes>

*)

PROPERTY long :ILongDateAndTimeAssertions
GET
END_GET
END_PROPERTY

(*

## Short summary
Returns the interface `ISimpleDateAndTimeAssertions` with assert statements for date and time types with 32 bit length

.. <legal notes>

legal notes
=================
| SPDX-FileCopyrightText: © 2022 ekvip automation GmbH <info@ekvip.de>
| SPDX-License-Identifier: Apache-2.0
| For details check: Apache-2.0_

.. _Apache-2.0: https://www.apache.org/licenses/LICENSE-2.0

.. </legal notes>



*)

PROPERTY simple :ISimpleDateAndTimeAssertions
GET
END_GET
END_PROPERTY

END_INTERFACE

// ---- Assertor/Assertions/FloatAssertions/interfaces/IFloatAssertions.TcIO
(*

## Short summary
This interface provides assert statements for floatings (``REAL`` and ``LREAL``)
For 32 bit floats (``REAL``) use `IFloatAssertions.single`
For 64 bit floats (``LREAL``) use `IFloatAssertions.double`

.. <legal notes>

legal notes
=================
| SPDX-FileCopyrightText: © 2022 ekvip automation GmbH <info@ekvip.de>
| SPDX-License-Identifier: Apache-2.0
| For details check: Apache-2.0_

.. _Apache-2.0: https://www.apache.org/licenses/LICENSE-2.0

.. </legal notes>



*)

INTERFACE IFloatAssertions EXTENDS __SYSTEM.IQueryInterface

(*

## Short summary
Returns the interface `ILrealAssertions` with assert statements for 64 bit floatings (``LREAL``)

.. <legal notes>

legal notes
=================
| SPDX-FileCopyrightText: © 2022 ekvip automation GmbH <info@ekvip.de>
| SPDX-License-Identifier: Apache-2.0
| For details check: Apache-2.0_

.. _Apache-2.0: https://www.apache.org/licenses/LICENSE-2.0

.. </legal notes>

*)

PROPERTY double :ILrealAssertions
GET
END_GET
END_PROPERTY

(*

## Short summary
Returns the interface `IRealAssertions` with assert statements for 32 bit floatings (``REAL``)

.. <legal notes>

legal notes
=================
| SPDX-FileCopyrightText: © 2022 ekvip automation GmbH <info@ekvip.de>
| SPDX-License-Identifier: Apache-2.0
| For details check: Apache-2.0_

.. _Apache-2.0: https://www.apache.org/licenses/LICENSE-2.0

.. </legal notes>

*)

PROPERTY single :IRealAssertions
GET
END_GET
END_PROPERTY

END_INTERFACE

// ---- Assertor/Assertions/FloatAssertions/Lreal/interfaces/ILrealAssertions.TcIO
(*

## Short summary
This interface provides assert statements for 64 bit floatings (``LREAL``) 

.. <legal notes>

legal notes
=================
| SPDX-FileCopyrightText: © 2022 ekvip automation GmbH <info@ekvip.de>
| SPDX-License-Identifier: Apache-2.0
| For details check: Apache-2.0_

.. _Apache-2.0: https://www.apache.org/licenses/LICENSE-2.0

.. </legal notes>



*)

INTERFACE ILrealAssertions EXTENDS __SYSTEM.IQueryInterface

(*

## Short summary
This assertion method checks if the current value is a number (NOT NaN)
for details check [IEEE 754](https://en.wikipedia.org/wiki/IEEE_754)


.. <legal notes>

legal notes
=================
| SPDX-FileCopyrightText: © 2023 ekvip automation GmbH <info@ekvip.de>
| SPDX-License-Identifier: Apache-2.0
| For details check: Apache-2.0_

.. _Apache-2.0: https://www.apache.org/licenses/LICENSE-2.0

.. </legal notes>



*)

METHOD valueIsANumber
VAR_INPUT
	(* current value to check *)
	currentValue	:LREAL;
	(* message if the assertion is false *)
	message			:AssertMessage;
END_VAR
END_METHOD

(*

## Short summary
This assertion method checks if the current value is equal to the expected value

**Attention:** 
	Nothing is equal to NaN, that means if ``currentValue`` OR ``expectedValue`` OR ``tolerance``
	is NaN then is the assertion false. For details check `IEEE 754`_

**Attention:** 
	infinity is equal to infinity and -infinity is equal to -infinity, that means if
	``currentValue`` AND ``expectedValue`` have the value infinity 
	OR ``currentValue`` AND ``expectedValue`` have the value -infinity
	the assertion is TRUE. For details check `IEEE 754`_

**Attention:** 
	If ``tolerance`` has the value infinity or -infinity and 
	``currentValue`` is not NaN and ``expectedValue`` is not NaN
	then is the assertion true. for details check [IEEE 754](https://en.wikipedia.org/wiki/IEEE_754)


.. <legal notes>

legal notes
=================
| SPDX-FileCopyrightText: © 2022 ekvip automation GmbH <info@ekvip.de>
| SPDX-License-Identifier: Apache-2.0
| For details check: Apache-2.0_

.. _Apache-2.0: https://www.apache.org/licenses/LICENSE-2.0

.. </legal notes>



*)

METHOD valueIsEqualTo
VAR_INPUT
	(* current value to check *)
	currentValue	:LREAL;
	(* expected value to compare *)
	expectedValue	:LREAL;
	(* tolerance to compensate twiddling floats, it has no sign *)
	tolerance		:LREAL;
	(* message if the assertion is false *)
	message			:AssertMessage;
END_VAR
END_METHOD

(*

## Short summary
This assertion method checks if the current value is finite
(NOT (infinity OR -inifinity)), for details check [IEEE 754](https://en.wikipedia.org/wiki/IEEE_754)


.. <legal notes>

legal notes
=================
| SPDX-FileCopyrightText: © 2023 ekvip automation GmbH <info@ekvip.de>
| SPDX-License-Identifier: Apache-2.0
| For details check: Apache-2.0_

.. _Apache-2.0: https://www.apache.org/licenses/LICENSE-2.0

.. </legal notes>



*)

METHOD valueIsFinite
VAR_INPUT
	(* current value to check *)
	currentValue	:LREAL;
	(* message if the assertion is false *)
	message			:AssertMessage;
END_VAR
END_METHOD

(*

## Short summary
This assertion method checks if the current value is greater than the less value

**Attention:** 
	Any comparsion to NaN is ``FALSE`` that means if ``currentValue`` OR ``lessValue``
	is NaN then is the assertion false.
	For details check `IEEE 754`_ and the truth table below.

**Attention:** 
	Every number is smaller than infinity except infinity, it's equal.
	Every number is greater than -infinity except -infinity, it's equal.
	For details check [IEEE 754](https://en.wikipedia.org/wiki/IEEE_754) and the truth table below.


truth table for special values
===============================
+----------------------+-------------------+---------------+
| **``currentValue``** | **``lessValue``** | **assertion** |
+======================+===================+===============+
| NaN                  | Any value         | FALSE         |
+----------------------+-------------------+---------------+
| Any value            | NaN               | FALSE         |
+----------------------+-------------------+---------------+
| infinity             | NOT NaN           | TRUE          |
|                      | NOT infinity      |               |
+----------------------+-------------------+---------------+
| -infinity             | Any value         | FALSE         |
+----------------------+-------------------+---------------+
| Any value            | infinity          | FALSE         |
+----------------------+-------------------+---------------+
| NOT NaN              | -inifinity        | TRUE          |
| NOT -infinity        |                   |               |
+----------------------+-------------------+---------------+

.. <legal notes>

legal notes
=================
| SPDX-FileCopyrightText: © 2022 ekvip automation GmbH <info@ekvip.de>
| SPDX-License-Identifier: Apache-2.0
| For details check: Apache-2.0_

.. _Apache-2.0: https://www.apache.org/licenses/LICENSE-2.0

.. </legal notes>



*)

METHOD valueIsGreaterThan
VAR_INPUT
	(* current value to check *)
	currentValue	:LREAL;
	(* less than lower limit *)
	lessValue		:LREAL;
	(* message if the assertion is false *)
	message			:AssertMessage;
END_VAR
END_METHOD

(*

## Short summary
This assertion method checks if the current value is infinite
(infinity OR -inifinity), for details check [IEEE 754](https://en.wikipedia.org/wiki/IEEE_754)


.. <legal notes>

legal notes
=================
| SPDX-FileCopyrightText: © 2023 ekvip automation GmbH <info@ekvip.de>
| SPDX-License-Identifier: Apache-2.0
| For details check: Apache-2.0_

.. _Apache-2.0: https://www.apache.org/licenses/LICENSE-2.0

.. </legal notes>



*)

METHOD valueIsInfinite
VAR_INPUT
	(* current value to check *)
	currentValue	:LREAL;
	(* message if the assertion is false *)
	message			:AssertMessage;
END_VAR
END_METHOD

(*

## Short summary
This assertion method checks if the current value is inside a limit

**Attention:** 
	limits are included: ``valueIsInRangeOf(3.0, 3.0, 3.0)`` is a true assertion

**Attention:** 
	Any comparsion to NaN is ``FALSE`` that means 
	if ``lowerLimit`` OR ``currentValue`` OR ``upperLimit``
	is NaN then is the assertion false.
	For details check `IEEE 754`_ and the truth table below.

**Attention:** 
	Every number is smaller than infinity except infinity, it's equal.
	Every number is greater than -infinity except -infinity, it's equal.
	For details check [IEEE 754](https://en.wikipedia.org/wiki/IEEE_754) and the truth table below.


truth table for special values
===============================
+--------------------+----------------------+--------------------+---------------+
| **``lowerLimit``** | **``currentValue``** | **``upperLimit``** | **assertion** |
+====================+======================+====================+===============+
| NaN                | Any value            | Any value          | FASLE         |
+--------------------+----------------------+--------------------+---------------+
| Any value          | NaN                  | Any value          | FALSE         |
+--------------------+----------------------+--------------------+---------------+
| Any value          | Any value            | NaN                | FALSE         |
+--------------------+----------------------+--------------------+---------------+
| -infinity          | NOT NaN              | infinity           | TRUE          |
+--------------------+----------------------+--------------------+---------------+
| infinity           | Any value            | -infinity          | FALSE         |
+--------------------+----------------------+--------------------+---------------+
| NOT -infinity      | -infinity            | Any value          | FALSE         |
+--------------------+----------------------+--------------------+---------------+
| Any value          | infinity             | NOT infinity       | FALSE         |
+--------------------+----------------------+--------------------+---------------+
| -infinity          | -infinity            | -infinity          | TRUE          |
+--------------------+----------------------+--------------------+---------------+
| infinity           | infinity             | infinity           | TRUE          |
+--------------------+----------------------+--------------------+---------------+
| -infinity          | NOT -infinity        | -infinity          | FALSE         |
+--------------------+----------------------+--------------------+---------------+
| infinity           | NOT infinity         | infinity           | FALSE         |
+--------------------+----------------------+--------------------+---------------+

.. <legal notes>

legal notes
=================
| SPDX-FileCopyrightText: © 2022 ekvip automation GmbH <info@ekvip.de>
| SPDX-License-Identifier: Apache-2.0
| For details check: Apache-2.0_

.. _Apache-2.0: https://www.apache.org/licenses/LICENSE-2.0

.. </legal notes>



*)

METHOD valueIsInRangeOf
VAR_INPUT
	(* lower limit for the current value *)
	lowerLimit		:LREAL;
	(* current value to check *)
	currentValue	:LREAL;
	(* upper limit for the current value *)
	upperLimit		:LREAL;
	(* message if the assertion is false *)
	message			:AssertMessage;
END_VAR
END_METHOD

(*

## Short summary
This assertion method checks if the current value is greater than the less value

**Attention:**
	Any comparsion to NaN is ``FALSE`` that means if ``currentValue`` OR ``greaterValue``
	is NaN then is the assertion false.
	For details check `IEEE 754`_ and the truth table below.

**Attention:**
	Every number is smaller than infinity except infinity, it's equal.
	Every number is greater than -infinity except -infinity, it's equal.
	For details check [IEEE 754](https://en.wikipedia.org/wiki/IEEE_754) and the truth table below.


truth table for special values
===============================
+----------------------+----------------------+---------------+
| **``currentValue``** | **``greaterValue``** | **assertion** |
+======================+======================+===============+
| NaN                  | Any value            | FASLE         |
+----------------------+----------------------+---------------+
| Any value            | NaN                  | FALSE         |
+----------------------+----------------------+---------------+
| infinity             | Any value            | FALSE         |
+----------------------+----------------------+---------------+
| -infinity             | NOT NaN              | TRUE          |
|                      | NOT -infinity        |               |
+----------------------+----------------------+---------------+
| NOT NaN              | infinity             | TRUE          |
| NOT infinity         |                      |               |
+----------------------+----------------------+---------------+

.. <legal notes>

legal notes
=================
| SPDX-FileCopyrightText: © 2022 ekvip automation GmbH <info@ekvip.de>
| SPDX-License-Identifier: Apache-2.0
| For details check: Apache-2.0_

.. _Apache-2.0: https://www.apache.org/licenses/LICENSE-2.0

.. </legal notes>



*)

METHOD valueIsLessThan
VAR_INPUT
	(* current value to check *)
	currentValue	:LREAL;
	(* greater than upper limit *)
	greaterValue	:LREAL;
	(* message if the assertion is false *)
	message			:AssertMessage;
END_VAR
END_METHOD

(*

## Short summary
This assertion method checks if the current value is less than or equal to the maximum value

**Attention:**
	Any comparsion to NaN is ``FALSE`` that means if ``currentValue`` OR ``maximumValue``
	is NaN then is the assertion false.
	For details check `IEEE 754`_ and the truth table below.

**Attention:**
	Every number is smaller than infinity except infinity, it's equal.
	Every number is greater than -infinity except -infinity, it's equal.
	For details check [IEEE 754](https://en.wikipedia.org/wiki/IEEE_754) and the truth table below.


truth table for special values
===============================
+----------------------+----------------------+---------------+
| **``currentValue``** | **``maximumValue``** | **assertion** |
+======================+======================+===============+
| NaN                  | Any value            | FASLE         |
+----------------------+----------------------+---------------+
| Any value            | NaN                  | FALSE         |
+----------------------+----------------------+---------------+
| NOT NaN              | infinity             | TRUE          |
+----------------------+----------------------+---------------+
| -infinity            | NOT NaN              | TRUE          |
+----------------------+----------------------+---------------+
| infinity             | NOT infinity         | FALSE         |
+----------------------+----------------------+---------------+
| NOT -infinity        | -infinity            | FALSE         |
+----------------------+----------------------+---------------+

.. <legal notes>

legal notes
=================
| SPDX-FileCopyrightText: © 2022 ekvip automation GmbH <info@ekvip.de>
| SPDX-License-Identifier: Apache-2.0
| For details check: Apache-2.0_

.. _Apache-2.0: https://www.apache.org/licenses/LICENSE-2.0

.. </legal notes>



*)

METHOD valueIsMax
VAR_INPUT
	(* current value to check *)
	currentValue	:LREAL;
	(* upper limit for the current value *)
	maximumValue	:LREAL;
	(* message if the assertion is false *)
	message			:AssertMessage;
END_VAR
END_METHOD

(*

## Short summary
This assertion method checks if the current value is greater than or equal to the minimum value

**Attention:**
	Any comparsion to NaN is ``FALSE`` that means if ``currentValue`` OR ``minimumValue``
	is NaN then is the assertion false.
	For details check `IEEE 754`_ and the truth table below.

**Attention:**
	Every number is smaller than infinity except infinity, it's equal.
	Every number is greater than -infinity except -infinity, it's equal.
	For details check [IEEE 754](https://en.wikipedia.org/wiki/IEEE_754) and the truth table below.


truth table for special values
===============================
+----------------------+----------------------+---------------+
| **``currentValue``** | **``minimumValue``** | **assertion** |
+======================+======================+===============+
| NaN                  | Any value            | FASLE         |
+----------------------+----------------------+---------------+
| Any value            | NaN                  | FALSE         |
+----------------------+----------------------+---------------+
| infinity             | NOT NaN              | TRUE          |
+----------------------+----------------------+---------------+
| NOT NaN              | -infinity            | TRUE          |
+----------------------+----------------------+---------------+
| -infinity            | NOT -infinity        | FALSE         |
+----------------------+----------------------+---------------+
| NOT infinity         | infinity             | FALSE         |
+----------------------+----------------------+---------------+

.. <legal notes>

legal notes
=================
| SPDX-FileCopyrightText: © 2022 ekvip automation GmbH <info@ekvip.de>
| SPDX-License-Identifier: Apache-2.0
| For details check: Apache-2.0_

.. _Apache-2.0: https://www.apache.org/licenses/LICENSE-2.0

.. </legal notes>



*)

METHOD valueIsMin
VAR_INPUT
	(* current value to check *)
	currentValue	:LREAL;
	(* lower limit for the current value *)
	minimumValue	:LREAL;
	(* message if the assertion is false *)
	message			:AssertMessage;
END_VAR
END_METHOD

(*

## Short summary
This assertion method checks if the current value is a not a number (NaN)
for details check [IEEE 754](https://en.wikipedia.org/wiki/IEEE_754)


.. <legal notes>

legal notes
=================
| SPDX-FileCopyrightText: © 2023 ekvip automation GmbH <info@ekvip.de>
| SPDX-License-Identifier: Apache-2.0
| For details check: Apache-2.0_

.. _Apache-2.0: https://www.apache.org/licenses/LICENSE-2.0

.. </legal notes>



*)

METHOD valueIsNaN
VAR_INPUT
	(* current value to check *)
	currentValue	:LREAL;
	(* message if the assertion is false *)
	message			:AssertMessage;
END_VAR
END_METHOD

(*

## Short summary
This assertion method checks if the current value is negative

**Attention:**
	Any comparsion to NaN is ``FALSE`` that means if ``currentValue``
	is NaN then is the assertion false.
	For details check `IEEE 754`_.

**Attention:**
	``currentValue`` has the value infinity means the assertion is false.
	``currentValue`` has the value -infinity means the assertion is true.
	``currentValue`` has the +0.0 means the assertion is false.
	``currentValue`` has the value -0.0 means the assertion is true.	
		For details check [IEEE 754](https://en.wikipedia.org/wiki/IEEE_754).


.. <legal notes>

legal notes
=================
| SPDX-FileCopyrightText: © 2022 ekvip automation GmbH <info@ekvip.de>
| SPDX-License-Identifier: Apache-2.0
| For details check: Apache-2.0_

.. _Apache-2.0: https://www.apache.org/licenses/LICENSE-2.0

.. </legal notes>



*)

METHOD valueIsNegative
VAR_INPUT
	(* current value to check *)
	currentValue	:LREAL;
	(* message if the assertion is false *)
	message			:AssertMessage;
END_VAR
END_METHOD

(*

## Short summary
This assertion method checks if the current value is negative infinite
(-infinity), for details check [IEEE 754](https://en.wikipedia.org/wiki/IEEE_754)


.. <legal notes>

legal notes
=================
| SPDX-FileCopyrightText: © 2023 ekvip automation GmbH <info@ekvip.de>
| SPDX-License-Identifier: Apache-2.0
| For details check: Apache-2.0_

.. _Apache-2.0: https://www.apache.org/licenses/LICENSE-2.0

.. </legal notes>



*)

METHOD valueIsNegativeInfinite
VAR_INPUT
	(* current value to check *)
	currentValue	:LREAL;
	(* message if the assertion is false *)
	message			:AssertMessage;
END_VAR
END_METHOD

(*

## Short summary
This assertion method checks if the current value is -0.0
for details check [IEEE 754](https://en.wikipedia.org/wiki/IEEE_754)


.. <legal notes>

legal notes
=================
| SPDX-FileCopyrightText: © 2023 ekvip automation GmbH <info@ekvip.de>
| SPDX-License-Identifier: Apache-2.0
| For details check: Apache-2.0_

.. _Apache-2.0: https://www.apache.org/licenses/LICENSE-2.0

.. </legal notes>



*)

METHOD valueIsNegativeZero
VAR_INPUT
	(* current value to check *)
	currentValue	:LREAL;
	(* message if the assertion is false *)
	message			:AssertMessage;
END_VAR
END_METHOD

(*

## Short summary
This assertion method checks if the current value is a normal number (not subnormal)
for details check [IEEE 754](https://en.wikipedia.org/wiki/IEEE_754)


.. <legal notes>

legal notes
=================
| SPDX-FileCopyrightText: © 2023 ekvip automation GmbH <info@ekvip.de>
| SPDX-License-Identifier: Apache-2.0
| For details check: Apache-2.0_

.. _Apache-2.0: https://www.apache.org/licenses/LICENSE-2.0

.. </legal notes>



*)

METHOD valueIsNormal
VAR_INPUT
	(* current value to check *)
	currentValue	:LREAL;
	(* message if the assertion is false *)
	message			:AssertMessage;
END_VAR
END_METHOD

(*

## Short summary
This assertion method checks if the current value is not equal to the unexpected value

**Attention:** 
	Nothing is equal to NaN, that means if ``currentValue`` OR ``unexpectedValue`` OR ``tolerance``
	is NaN then is the assertion true. For details check `IEEE 754`_

**Attention:** 
	infinity is equal to infinity and -infinity is equal to -infinity, that means if
	``currentValue`` AND ``unexpectedValue`` have the value infinity 
	OR ``currentValue`` AND ``unexpectedValue`` have the value -infinity
	the assertion is false. For details check `IEEE 754`_

**Attention:** 
	If ``tolerance`` has the value infinity or -infinity and 
	``currentValue`` is not NaN and ``unexpectedValue`` is not NaN
	then is the assertion false. for details check [IEEE 754](https://en.wikipedia.org/wiki/IEEE_754)


.. <legal notes>

legal notes
=================
| SPDX-FileCopyrightText: © 2022 ekvip automation GmbH <info@ekvip.de>
| SPDX-License-Identifier: Apache-2.0
| For details check: Apache-2.0_

.. _Apache-2.0: https://www.apache.org/licenses/LICENSE-2.0

.. </legal notes>



*)

METHOD valueIsNotEqualTo
VAR_INPUT
	(* current value to check *)
	currentValue	:LREAL;
	(* unexpected value to compare *)
	unexpectedValue	:LREAL;
	(* tolerance to compensate twiddling floats, it has no sign *)
	tolerance		:LREAL;
	(* message if the assertion is false *)
	message			:AssertMessage;
END_VAR
END_METHOD

(*

## Short summary
This assertion method checks if the current value is not negative infinite
NOT (-infinity), for details check [IEEE 754](https://en.wikipedia.org/wiki/IEEE_754)


.. <legal notes>

legal notes
=================
| SPDX-FileCopyrightText: © 2023 ekvip automation GmbH <info@ekvip.de>
| SPDX-License-Identifier: Apache-2.0
| For details check: Apache-2.0_

.. _Apache-2.0: https://www.apache.org/licenses/LICENSE-2.0

.. </legal notes>



*)

METHOD valueIsNotNegativeInfinite
VAR_INPUT
	(* current value to check *)
	currentValue	:LREAL;
	(* message if the assertion is false *)
	message			:AssertMessage;
END_VAR
END_METHOD

(*

## Short summary
This assertion method checks if the current value is not positive infinite
NOT (infinity), for details check [IEEE 754](https://en.wikipedia.org/wiki/IEEE_754)


.. <legal notes>

legal notes
=================
| SPDX-FileCopyrightText: © 2023 ekvip automation GmbH <info@ekvip.de>
| SPDX-License-Identifier: Apache-2.0
| For details check: Apache-2.0_

.. _Apache-2.0: https://www.apache.org/licenses/LICENSE-2.0

.. </legal notes>



*)

METHOD valueIsNotPositiveInfinite
VAR_INPUT
	(* current value to check *)
	currentValue	:LREAL;
	(* message if the assertion is false *)
	message			:AssertMessage;
END_VAR
END_METHOD

(*

## Short summary
This assertion method checks if the current value is a non special number
(NOT (NaN OR infinity OR -inifinity)), for details check [IEEE 754](https://en.wikipedia.org/wiki/IEEE_754)


.. <legal notes>

legal notes
=================
| SPDX-FileCopyrightText: © 2023 ekvip automation GmbH <info@ekvip.de>
| SPDX-License-Identifier: Apache-2.0
| For details check: Apache-2.0_

.. _Apache-2.0: https://www.apache.org/licenses/LICENSE-2.0

.. </legal notes>



*)

METHOD valueIsNotSpecial
VAR_INPUT
	(* current value to check *)
	currentValue	:LREAL;
	(* message if the assertion is false *)
	message			:AssertMessage;
END_VAR
END_METHOD

(*

## Short summary
This assertion method checks if the current value is positve

**Attention:**
	Any comparsion to NaN is ``FALSE`` that means if ``currentValue``
	is NaN then is the assertion false.
	For details check `IEEE 754`_.

**Attention:**
	``currentValue`` has the value infinity means the assertion is true.
	``currentValue`` has the value -infinity means the assertion is false.
	``currentValue`` has the +0.0 means the assertion is true.
	``currentValue`` has the value -0.0 means the assertion is false.	
		For details check [IEEE 754](https://en.wikipedia.org/wiki/IEEE_754).


.. <legal notes>

legal notes
=================
| SPDX-FileCopyrightText: © 2022 ekvip automation GmbH <info@ekvip.de>
| SPDX-License-Identifier: Apache-2.0
| For details check: Apache-2.0_

.. _Apache-2.0: https://www.apache.org/licenses/LICENSE-2.0

.. </legal notes>



*)

METHOD valueIsPositive
VAR_INPUT
	(* current value to check *)
	currentValue	:LREAL;
	(* message if the assertion is false *)
	message			:AssertMessage;
END_VAR
END_METHOD

(*

## Short summary
This assertion method checks if the current value is positive infinite
(infinity), for details check [IEEE 754](https://en.wikipedia.org/wiki/IEEE_754)


.. <legal notes>

legal notes
=================
| SPDX-FileCopyrightText: © 2023 ekvip automation GmbH <info@ekvip.de>
| SPDX-License-Identifier: Apache-2.0
| For details check: Apache-2.0_

.. _Apache-2.0: https://www.apache.org/licenses/LICENSE-2.0

.. </legal notes>



*)

METHOD valueIsPositiveInfinite
VAR_INPUT
	(* current value to check *)
	currentValue	:LREAL;
	(* message if the assertion is false *)
	message			:AssertMessage;
END_VAR
END_METHOD

(*

## Short summary
This assertion method checks if the current value is +0.0
for details check [IEEE 754](https://en.wikipedia.org/wiki/IEEE_754)


.. <legal notes>

legal notes
=================
| SPDX-FileCopyrightText: © 2023 ekvip automation GmbH <info@ekvip.de>
| SPDX-License-Identifier: Apache-2.0
| For details check: Apache-2.0_

.. _Apache-2.0: https://www.apache.org/licenses/LICENSE-2.0

.. </legal notes>



*)

METHOD valueIsPositiveZero
VAR_INPUT
	(* current value to check *)
	currentValue	:LREAL;
	(* message if the assertion is false *)
	message			:AssertMessage;
END_VAR
END_METHOD

(*

## Short summary
This assertion method checks if the current value is a special
(NaN OR infinity OR -inifinity), for details check [IEEE 754](https://en.wikipedia.org/wiki/IEEE_754)


.. <legal notes>

legal notes
=================
| SPDX-FileCopyrightText: © 2023 ekvip automation GmbH <info@ekvip.de>
| SPDX-License-Identifier: Apache-2.0
| For details check: Apache-2.0_

.. _Apache-2.0: https://www.apache.org/licenses/LICENSE-2.0

.. </legal notes>



*)

METHOD valueIsSpecial
VAR_INPUT
	(* current value to check *)
	currentValue	:LREAL;
	(* message if the assertion is false *)
	message			:AssertMessage;
END_VAR
END_METHOD

(*

## Short summary
This assertion method checks if the current value is a subnormal number
for details check [IEEE 754](https://en.wikipedia.org/wiki/IEEE_754)


.. <legal notes>

legal notes
=================
| SPDX-FileCopyrightText: © 2023 ekvip automation GmbH <info@ekvip.de>
| SPDX-License-Identifier: Apache-2.0
| For details check: Apache-2.0_

.. _Apache-2.0: https://www.apache.org/licenses/LICENSE-2.0

.. </legal notes>



*)

METHOD valueIsSubnormal
VAR_INPUT
	(* current value to check *)
	currentValue	:LREAL;
	(* message if the assertion is false *)
	message			:AssertMessage;
END_VAR
END_METHOD

END_INTERFACE

// ---- Assertor/Assertions/FloatAssertions/Real/interfaces/IRealAssertions.TcIO
(*

## Short summary
This interface provides assert statements for 32 bit floatings (``REAL``)

.. <legal notes>

legal notes
=================
| SPDX-FileCopyrightText: © 2022 ekvip automation GmbH <info@ekvip.de>
| SPDX-License-Identifier: Apache-2.0
| For details check: Apache-2.0_

.. _Apache-2.0: https://www.apache.org/licenses/LICENSE-2.0

.. </legal notes>



*)

INTERFACE IRealAssertions EXTENDS __SYSTEM.IQueryInterface

(*

## Short summary
This assertion method checks if the current value is a number (NOT NaN)
for details check [IEEE 754](https://en.wikipedia.org/wiki/IEEE_754)


.. <legal notes>

legal notes
=================
| SPDX-FileCopyrightText: © 2023 ekvip automation GmbH <info@ekvip.de>
| SPDX-License-Identifier: Apache-2.0
| For details check: Apache-2.0_

.. _Apache-2.0: https://www.apache.org/licenses/LICENSE-2.0

.. </legal notes>



*)

METHOD valueIsANumber
VAR_INPUT
	(* current value to check *)
	currentValue	:REAL;
	(* message if the assertion is false *)
	message			:AssertMessage;
END_VAR
END_METHOD

(*

## Short summary
This assertion method checks if the current value is equal to the expected value

**Attention:** 
	Nothing is equal to NaN, that means if ``currentValue`` OR ``expectedValue`` OR ``tolerance``
	is NaN then is the assertion false. For details check `IEEE 754`_

**Attention:** 
	infinity is equal to infinity and -infinity is equal to -infinity, that means if
	``currentValue`` AND ``expectedValue`` have the value infinity 
	OR ``currentValue`` AND ``expectedValue`` have the value -infinity
	the assertion is TRUE. For details check `IEEE 754`_

**Attention:** 
	If ``tolerance`` has the value infinity or -infinity and 
	``currentValue`` is not NaN and ``expectedValue`` is not NaN
	then is the assertion true. for details check [IEEE 754](https://en.wikipedia.org/wiki/IEEE_754)


.. <legal notes>

legal notes
=================
| SPDX-FileCopyrightText: © 2022 ekvip automation GmbH <info@ekvip.de>
| SPDX-License-Identifier: Apache-2.0
| For details check: Apache-2.0_

.. _Apache-2.0: https://www.apache.org/licenses/LICENSE-2.0

.. </legal notes>



*)

METHOD valueIsEqualTo
VAR_INPUT
	(* current value to check *)
	currentValue	:REAL;
	(* expected value to compare *)
	expectedValue	:REAL;
	(* tolerance to compensate twiddling floats *)
	tolerance		:REAL;
	(* message if the assertion is false *)
	message			:AssertMessage;
END_VAR
END_METHOD

(*

## Short summary
This assertion method checks if the current value is finite
(NOT (infinity OR -inifinity)), for details check [IEEE 754](https://en.wikipedia.org/wiki/IEEE_754)


.. <legal notes>

legal notes
=================
| SPDX-FileCopyrightText: © 2023 ekvip automation GmbH <info@ekvip.de>
| SPDX-License-Identifier: Apache-2.0
| For details check: Apache-2.0_

.. _Apache-2.0: https://www.apache.org/licenses/LICENSE-2.0

.. </legal notes>



*)

METHOD valueIsFinite
VAR_INPUT
	(* current value to check *)
	currentValue	:REAL;
	(* message if the assertion is false *)
	message			:AssertMessage;
END_VAR
END_METHOD

(*

## Short summary
This assertion method checks if the current value is greater than the less value

**Attention:** 
	Any comparsion to NaN is ``FALSE`` that means if ``currentValue`` OR ``lessValue``
	is NaN then is the assertion false.
	For details check `IEEE 754`_ and the truth table below.

**Attention:** 
	Every number is smaller than infinity except infinity, it's equal.
	Every number is greater than -infinity except -infinity, it's equal.
	For details check [IEEE 754](https://en.wikipedia.org/wiki/IEEE_754) and the truth table below.


truth table for special values
===============================
+----------------------+-------------------+---------------+
| **``currentValue``** | **``lessValue``** | **assertion** |
+======================+===================+===============+
| NaN                  | Any value         | FASLE         |
+----------------------+-------------------+---------------+
| Any value            | NaN               | FALSE         |
+----------------------+-------------------+---------------+
| infinity             | NOT NaN           | TRUE          |
|                      | NOT infinity      |               |
+----------------------+-------------------+---------------+
| -infinity             | Any value         | FALSE         |
+----------------------+-------------------+---------------+
| Any value            | infinity          | FALSE         |
+----------------------+-------------------+---------------+
| NOT NaN              | -inifinity        | TRUE          |
| NOT -infinity        |                   |               |
+----------------------+-------------------+---------------+

.. <legal notes>

legal notes
=================
| SPDX-FileCopyrightText: © 2022 ekvip automation GmbH <info@ekvip.de>
| SPDX-License-Identifier: Apache-2.0
| For details check: Apache-2.0_

.. _Apache-2.0: https://www.apache.org/licenses/LICENSE-2.0

.. </legal notes>



*)

METHOD valueIsGreaterThan
VAR_INPUT
	(* current value to check *)
	currentValue	:REAL;
	(* less than lower limit *)
	lessValue		:REAL;
	(* message if the assertion is false *)
	message			:AssertMessage;
END_VAR
END_METHOD

(*

## Short summary
This assertion method checks if the current value is infinite
(infinity OR -inifinity), for details check [IEEE 754](https://en.wikipedia.org/wiki/IEEE_754)


.. <legal notes>

legal notes
=================
| SPDX-FileCopyrightText: © 2023 ekvip automation GmbH <info@ekvip.de>
| SPDX-License-Identifier: Apache-2.0
| For details check: Apache-2.0_

.. _Apache-2.0: https://www.apache.org/licenses/LICENSE-2.0

.. </legal notes>



*)

METHOD valueIsInfinite
VAR_INPUT
	(* current value to check *)
	currentValue	:REAL;
	(* message if the assertion is false *)
	message			:AssertMessage;
END_VAR
END_METHOD

(*

## Short summary
This assertion method checks if the current value is inside a limit

**Attention:** 
	limits are included: ``valueIsInRangeOf(3.0, 3.0, 3.0)`` is a true assertion

**Attention:** 
	Any comparsion to NaN is ``FALSE`` that means 
	if ``lowerLimit`` OR ``currentValue`` OR ``upperLimit``
	is NaN then is the assertion false.
	For details check `IEEE 754`_ and the truth table below.

**Attention:** 
	Every number is smaller than infinity except infinity, it's equal.
	Every number is greater than -infinity except -infinity, it's equal.
	For details check [IEEE 754](https://en.wikipedia.org/wiki/IEEE_754) and the truth table below.


truth table for special values
===============================
+--------------------+----------------------+--------------------+---------------+
| **``lowerLimit``** | **``currentValue``** | **``upperLimit``** | **assertion** |
+====================+======================+====================+===============+
| NaN                | Any value            | Any value          | FASLE         |
+--------------------+----------------------+--------------------+---------------+
| Any value          | NaN                  | Any value          | FALSE         |
+--------------------+----------------------+--------------------+---------------+
| Any value          | Any value            | NaN                | FALSE         |
+--------------------+----------------------+--------------------+---------------+
| -infinity          | NOT NaN              | infinity           | TRUE          |
+--------------------+----------------------+--------------------+---------------+
| infinity           | Any value            | -infinity          | FALSE         |
+--------------------+----------------------+--------------------+---------------+
| NOT -infinity      | -infinity            | Any value          | FALSE         |
+--------------------+----------------------+--------------------+---------------+
| Any value          | infinity             | NOT infinity       | FALSE         |
+--------------------+----------------------+--------------------+---------------+
| -infinity          | -infinity            | -infinity          | TRUE          |
+--------------------+----------------------+--------------------+---------------+
| infinity           | infinity             | infinity           | TRUE          |
+--------------------+----------------------+--------------------+---------------+
| -infinity          | NOT -infinity        | -infinity          | FALSE         |
+--------------------+----------------------+--------------------+---------------+
| infinity           | NOT infinity         | infinity           | FALSE         |
+--------------------+----------------------+--------------------+---------------+

.. <legal notes>

legal notes
=================
| SPDX-FileCopyrightText: © 2022 ekvip automation GmbH <info@ekvip.de>
| SPDX-License-Identifier: Apache-2.0
| For details check: Apache-2.0_

.. _Apache-2.0: https://www.apache.org/licenses/LICENSE-2.0

.. </legal notes>



*)

METHOD valueIsInRangeOf
VAR_INPUT
	(* lower limit for the current value *)
	lowerLimit		:REAL;
	(* current value to check *)
	currentValue	:REAL;
	(* upper limit for the current value *)
	upperLimit		:REAL;
	(* message if the assertion is false *)
	message			:AssertMessage;
END_VAR
END_METHOD

(*

## Short summary
This assertion method checks if the current value is greater than the less value

**Attention:**
	Any comparsion to NaN is ``FALSE`` that means if ``currentValue`` OR ``greaterValue``
	is NaN then is the assertion false.
	For details check `IEEE 754`_ and the truth table below.

**Attention:**
	Every number is smaller than infinity except infinity, it's equal.
	Every number is greater than -infinity except -infinity, it's equal.
	For details check [IEEE 754](https://en.wikipedia.org/wiki/IEEE_754) and the truth table below.


truth table for special values
===============================
+----------------------+----------------------+---------------+
| **``currentValue``** | **``greaterValue``** | **assertion** |
+======================+======================+===============+
| NaN                  | Any value            | FASLE         |
+----------------------+----------------------+---------------+
| Any value            | NaN                  | FALSE         |
+----------------------+----------------------+---------------+
| infinity             | Any value            | FALSE         |
+----------------------+----------------------+---------------+
| -infinity             | NOT NaN              | TRUE          |
|                      | NOT -infinity        |               |
+----------------------+----------------------+---------------+
| NOT NaN              | infinity             | TRUE          |
| NOT infinity         |                      |               |
+----------------------+----------------------+---------------+

.. <legal notes>

legal notes
=================
| SPDX-FileCopyrightText: © 2022 ekvip automation GmbH <info@ekvip.de>
| SPDX-License-Identifier: Apache-2.0
| For details check: Apache-2.0_

.. _Apache-2.0: https://www.apache.org/licenses/LICENSE-2.0

.. </legal notes>



*)

METHOD valueIsLessThan
VAR_INPUT
	(* current value to check *)
	currentValue	:REAL;
	(* greater than upper limit *)
	greaterValue	:REAL;
	(* message if the assertion is false *)
	message			:AssertMessage;
END_VAR
END_METHOD

(*

## Short summary
This assertion method checks if the current value is less than or equal to the maximum value

**Attention:**
	Any comparsion to NaN is ``FALSE`` that means if ``currentValue`` OR ``maximumValue``
	is NaN then is the assertion false.
	For details check `IEEE 754`_ and the truth table below.

**Attention:**
	Every number is smaller than infinity except infinity, it's equal.
	Every number is greater than -infinity except -infinity, it's equal.
	For details check [IEEE 754](https://en.wikipedia.org/wiki/IEEE_754) and the truth table below.


truth table for special values
===============================
+----------------------+----------------------+---------------+
| **``currentValue``** | **``maximumValue``** | **assertion** |
+======================+======================+===============+
| NaN                  | Any value            | FASLE         |
+----------------------+----------------------+---------------+
| Any value            | NaN                  | FALSE         |
+----------------------+----------------------+---------------+
| NOT NaN              | infinity             | TRUE          |
+----------------------+----------------------+---------------+
| -infinity            | NOT NaN              | TRUE          |
+----------------------+----------------------+---------------+
| infinity             | NOT infinity         | FALSE         |
+----------------------+----------------------+---------------+
| NOT -infinity        | -infinity            | FALSE         |
+----------------------+----------------------+---------------+

.. <legal notes>

legal notes
=================
| SPDX-FileCopyrightText: © 2022 ekvip automation GmbH <info@ekvip.de>
| SPDX-License-Identifier: Apache-2.0
| For details check: Apache-2.0_

.. _Apache-2.0: https://www.apache.org/licenses/LICENSE-2.0

.. </legal notes>



*)

METHOD valueIsMax
VAR_INPUT
	(* current value to check *)
	currentValue	:REAL;
	(* upper limit for the current value *)
	maximumValue	:REAL;
	(* message if the assertion is false *)
	message			:AssertMessage;
END_VAR
END_METHOD

(*

## Short summary
This assertion method checks if the current value is greater than or equal to the minimum value

**Attention:**
	Any comparsion to NaN is ``FALSE`` that means if ``currentValue`` OR ``minimumValue``
	is NaN then is the assertion false.
	For details check `IEEE 754`_ and the truth table below.

**Attention:**
	Every number is smaller than infinity except infinity, it's equal.
	Every number is greater than -infinity except -infinity, it's equal.
	For details check [IEEE 754](https://en.wikipedia.org/wiki/IEEE_754) and the truth table below.


truth table for special values
===============================
+----------------------+----------------------+---------------+
| **``currentValue``** | **``minimumValue``** | **assertion** |
+======================+======================+===============+
| NaN                  | Any value            | FASLE         |
+----------------------+----------------------+---------------+
| Any value            | NaN                  | FALSE         |
+----------------------+----------------------+---------------+
| infinity             | NOT NaN              | TRUE          |
+----------------------+----------------------+---------------+
| NOT NaN              | -infinity            | TRUE          |
+----------------------+----------------------+---------------+
| -infinity            | NOT -infinity        | FALSE         |
+----------------------+----------------------+---------------+
| NOT infinity         | infinity             | FALSE         |
+----------------------+----------------------+---------------+

.. <legal notes>

legal notes
=================
| SPDX-FileCopyrightText: © 2022 ekvip automation GmbH <info@ekvip.de>
| SPDX-License-Identifier: Apache-2.0
| For details check: Apache-2.0_

.. _Apache-2.0: https://www.apache.org/licenses/LICENSE-2.0

.. </legal notes>



*)

METHOD valueIsMin
VAR_INPUT
	(* current value to check *)
	currentValue	:REAL;
	(* lower limit for the current value *)
	minimumValue	:REAL;
	(* message if the assertion is false *)
	message			:AssertMessage;
END_VAR
END_METHOD

(*

## Short summary
This assertion method checks if the current value is a not a number (NaN)
for details check [IEEE 754](https://en.wikipedia.org/wiki/IEEE_754)


.. <legal notes>

legal notes
=================
| SPDX-FileCopyrightText: © 2023 ekvip automation GmbH <info@ekvip.de>
| SPDX-License-Identifier: Apache-2.0
| For details check: Apache-2.0_

.. _Apache-2.0: https://www.apache.org/licenses/LICENSE-2.0

.. </legal notes>



*)

METHOD valueIsNaN
VAR_INPUT
	(* current value to check *)
	currentValue	:REAL;
	(* message if the assertion is false *)
	message			:AssertMessage;
END_VAR
END_METHOD

(*

## Short summary
This assertion method checks if the current value is negative

**Attention:**
	Any comparsion to NaN is ``FALSE`` that means if ``currentValue``
	is NaN then is the assertion false.
	For details check `IEEE 754`_.

**Attention:**
	``currentValue`` has the value infinity means the assertion is false.
	``currentValue`` has the value -infinity means the assertion is true.
	``currentValue`` has the +0.0 means the assertion is false.
	``currentValue`` has the value -0.0 means the assertion is true.	
		For details check [IEEE 754](https://en.wikipedia.org/wiki/IEEE_754).


.. <legal notes>

legal notes
=================
| SPDX-FileCopyrightText: © 2022 ekvip automation GmbH <info@ekvip.de>
| SPDX-License-Identifier: Apache-2.0
| For details check: Apache-2.0_

.. _Apache-2.0: https://www.apache.org/licenses/LICENSE-2.0

.. </legal notes>



*)

METHOD valueIsNegative
VAR_INPUT
	(* current value to check *)
	currentValue	:REAL;
	(* message if the assertion is false *)
	message			:AssertMessage;
END_VAR
END_METHOD

(*

## Short summary
This assertion method checks if the current value is negative infinite
(-infinity), for details check [IEEE 754](https://en.wikipedia.org/wiki/IEEE_754)


.. <legal notes>

legal notes
=================
| SPDX-FileCopyrightText: © 2023 ekvip automation GmbH <info@ekvip.de>
| SPDX-License-Identifier: Apache-2.0
| For details check: Apache-2.0_

.. _Apache-2.0: https://www.apache.org/licenses/LICENSE-2.0

.. </legal notes>



*)

METHOD valueIsNegativeInfinite
VAR_INPUT
	(* current value to check *)
	currentValue	:REAL;
	(* message if the assertion is false *)
	message			:AssertMessage;
END_VAR
END_METHOD

(*

## Short summary
This assertion method checks if the current value is +0.0
for details check [IEEE 754](https://en.wikipedia.org/wiki/IEEE_754)


.. <legal notes>

legal notes
=================
| SPDX-FileCopyrightText: © 2023 ekvip automation GmbH <info@ekvip.de>
| SPDX-License-Identifier: Apache-2.0
| For details check: Apache-2.0_

.. _Apache-2.0: https://www.apache.org/licenses/LICENSE-2.0

.. </legal notes>



*)

METHOD valueIsNegativeZero
VAR_INPUT
	(* current value to check *)
	currentValue	:REAL;
	(* message if the assertion is false *)
	message			:AssertMessage;
END_VAR
END_METHOD

(*

## Short summary
This assertion method checks if the current value is a normal number (not subnormal)
for details check [IEEE 754](https://en.wikipedia.org/wiki/IEEE_754)


.. <legal notes>

legal notes
=================
| SPDX-FileCopyrightText: © 2023 ekvip automation GmbH <info@ekvip.de>
| SPDX-License-Identifier: Apache-2.0
| For details check: Apache-2.0_

.. _Apache-2.0: https://www.apache.org/licenses/LICENSE-2.0

.. </legal notes>



*)

METHOD valueIsNormal
VAR_INPUT
	(* current value to check *)
	currentValue	:REAL;
	(* message if the assertion is false *)
	message			:AssertMessage;
END_VAR
END_METHOD

(*

## Short summary
This assertion method checks if the current value is not equal to the unexpected value

**Attention:** 
	Nothing is equal to NaN, that means if ``currentValue`` OR ``unexpectedValue`` OR ``tolerance``
	is NaN then is the assertion true. For details check `IEEE 754`_

**Attention:** 
	infinity is equal to infinity and -infinity is equal to -infinity, that means if
	``currentValue`` AND ``unexpectedValue`` have the value infinity 
	OR ``currentValue`` AND ``unexpectedValue`` have the value -infinity
	the assertion is false. For details check `IEEE 754`_

**Attention:** 
	If ``tolerance`` has the value infinity or -infinity and 
	``currentValue`` is not NaN and ``unexpectedValue`` is not NaN
	then is the assertion false. for details check [IEEE 754](https://en.wikipedia.org/wiki/IEEE_754)


.. <legal notes>

legal notes
=================
| SPDX-FileCopyrightText: © 2022 ekvip automation GmbH <info@ekvip.de>
| SPDX-License-Identifier: Apache-2.0
| For details check: Apache-2.0_

.. _Apache-2.0: https://www.apache.org/licenses/LICENSE-2.0

.. </legal notes>



*)

METHOD valueIsNotEqualTo
VAR_INPUT
	(* current value to check *)
	currentValue	:REAL;
	(* unexpected value to compare *)
	unexpectedValue	:REAL;
	(* tolerance to compensate twiddling floats *)
	tolerance		:REAL;
	(* message if the assertion is false *)
	message			:AssertMessage;
END_VAR
END_METHOD

(*

## Short summary
This assertion method checks if the current value is not negative infinite
NOT (-infinity), for details check [IEEE 754](https://en.wikipedia.org/wiki/IEEE_754)


.. <legal notes>

legal notes
=================
| SPDX-FileCopyrightText: © 2023 ekvip automation GmbH <info@ekvip.de>
| SPDX-License-Identifier: Apache-2.0
| For details check: Apache-2.0_

.. _Apache-2.0: https://www.apache.org/licenses/LICENSE-2.0

.. </legal notes>



*)

METHOD valueIsNotNegativeInfinite
VAR_INPUT
	(* current value to check *)
	currentValue	:REAL;
	(* message if the assertion is false *)
	message			:AssertMessage;
END_VAR
END_METHOD

(*

## Short summary
This assertion method checks if the current value is not positive infinite
NOT (infinity), for details check [IEEE 754](https://en.wikipedia.org/wiki/IEEE_754)


.. <legal notes>

legal notes
=================
| SPDX-FileCopyrightText: © 2023 ekvip automation GmbH <info@ekvip.de>
| SPDX-License-Identifier: Apache-2.0
| For details check: Apache-2.0_

.. _Apache-2.0: https://www.apache.org/licenses/LICENSE-2.0

.. </legal notes>



*)

METHOD valueIsNotPositiveInfinite
VAR_INPUT
	(* current value to check *)
	currentValue	:REAL;
	(* message if the assertion is false *)
	message			:AssertMessage;
END_VAR
END_METHOD

(*

## Short summary
This assertion method checks if the current value is a non special number
(NOT (NaN OR infinity OR -inifinity)), for details check [IEEE 754](https://en.wikipedia.org/wiki/IEEE_754)


.. <legal notes>

legal notes
=================
| SPDX-FileCopyrightText: © 2023 ekvip automation GmbH <info@ekvip.de>
| SPDX-License-Identifier: Apache-2.0
| For details check: Apache-2.0_

.. _Apache-2.0: https://www.apache.org/licenses/LICENSE-2.0

.. </legal notes>



*)

METHOD valueIsNotSpecial
VAR_INPUT
	(* current value to check *)
	currentValue	:REAL;
	(* message if the assertion is false *)
	message			:AssertMessage;
END_VAR
END_METHOD

(*

## Short summary
This assertion method checks if the current value is positve

**Attention:**
	Any comparsion to NaN is ``FALSE`` that means if ``currentValue``
	is NaN then is the assertion false.
	For details check `IEEE 754`_.

**Attention:**
	``currentValue`` has the value infinity means the assertion is true.
	``currentValue`` has the value -infinity means the assertion is false.
	``currentValue`` has the +0.0 means the assertion is true.
	``currentValue`` has the value -0.0 means the assertion is false.	
		For details check [IEEE 754](https://en.wikipedia.org/wiki/IEEE_754).


.. <legal notes>

legal notes
=================
| SPDX-FileCopyrightText: © 2022 ekvip automation GmbH <info@ekvip.de>
| SPDX-License-Identifier: Apache-2.0
| For details check: Apache-2.0_

.. _Apache-2.0: https://www.apache.org/licenses/LICENSE-2.0

.. </legal notes>



*)

METHOD valueIsPositive
VAR_INPUT
	(* current value to check *)
	currentValue	:REAL;
	(* message if the assertion is false *)
	message			:AssertMessage;
END_VAR
END_METHOD

(*

## Short summary
This assertion method checks if the current value is positive infinite
(infinity), for details check [IEEE 754](https://en.wikipedia.org/wiki/IEEE_754)


.. <legal notes>

legal notes
=================
| SPDX-FileCopyrightText: © 2023 ekvip automation GmbH <info@ekvip.de>
| SPDX-License-Identifier: Apache-2.0
| For details check: Apache-2.0_

.. _Apache-2.0: https://www.apache.org/licenses/LICENSE-2.0

.. </legal notes>



*)

METHOD valueIsPositiveInfinite
VAR_INPUT
	(* current value to check *)
	currentValue	:REAL;
	(* message if the assertion is false *)
	message			:AssertMessage;
END_VAR
END_METHOD

(*

## Short summary
This assertion method checks if the current value is -0.0
for details check [IEEE 754](https://en.wikipedia.org/wiki/IEEE_754)


.. <legal notes>

legal notes
=================
| SPDX-FileCopyrightText: © 2023 ekvip automation GmbH <info@ekvip.de>
| SPDX-License-Identifier: Apache-2.0
| For details check: Apache-2.0_

.. _Apache-2.0: https://www.apache.org/licenses/LICENSE-2.0

.. </legal notes>



*)

METHOD valueIsPositiveZero
VAR_INPUT
	(* current value to check *)
	currentValue	:REAL;
	(* message if the assertion is false *)
	message			:AssertMessage;
END_VAR
END_METHOD

(*

## Short summary
This assertion method checks if the current value is a special
(NaN OR infinity OR -inifinity), for details check [IEEE 754](https://en.wikipedia.org/wiki/IEEE_754)


.. <legal notes>

legal notes
=================
| SPDX-FileCopyrightText: © 2023 ekvip automation GmbH <info@ekvip.de>
| SPDX-License-Identifier: Apache-2.0
| For details check: Apache-2.0_

.. _Apache-2.0: https://www.apache.org/licenses/LICENSE-2.0

.. </legal notes>



*)

METHOD valueIsSpecial
VAR_INPUT
	(* current value to check *)
	currentValue	:REAL;
	(* message if the assertion is false *)
	message			:AssertMessage;
END_VAR
END_METHOD

(*

## Short summary
This assertion method checks if the current value is a subnormal number
for details check [IEEE 754](https://en.wikipedia.org/wiki/IEEE_754)


.. <legal notes>

legal notes
=================
| SPDX-FileCopyrightText: © 2023 ekvip automation GmbH <info@ekvip.de>
| SPDX-License-Identifier: Apache-2.0
| For details check: Apache-2.0_

.. _Apache-2.0: https://www.apache.org/licenses/LICENSE-2.0

.. </legal notes>



*)

METHOD valueIsSubnormal
VAR_INPUT
	(* current value to check *)
	currentValue	:REAL;
	(* message if the assertion is false *)
	message			:AssertMessage;
END_VAR
END_METHOD

END_INTERFACE

// ---- Assertor/Assertions/IntegerAssertions/interfaces/IIntegerAssertions.TcIO
(*

## Short summary
This interface provides assert statements for signed/unsigned integers from 8~64 bit length 
For signed integers use `IIntergerAssertions.signed`
For unsigned integers use `IIntergerAssertions.unsigned`

.. <legal notes>

legal notes
=================
| SPDX-FileCopyrightText: © 2022 ekvip automation GmbH <info@ekvip.de>
| SPDX-License-Identifier: Apache-2.0
| For details check: Apache-2.0_

